	MFD_NPBSS_6_damper_open AT%I* : BOOL;
	MFD_NPBSS_6_damper_close AT%I* : BOOL;

	MFD_NPBSS_7_damper_open AT%I* : BOOL;
	MFD_NPBSS_7_damper_close AT%I* : BOOL;

	MFD_NPBSS_8_damper_open AT%I* : BOOL;
	MFD_NPBSS_8_damper_close AT%I* : BOOL;

	MFD_NPBSS_9_damper_open AT%I* : BOOL;
	MFD_NPBSS_9_damper_close AT%I* : BOOL;

	MFD_NPBSS_10_damper_open AT%I* : BOOL;
	MFD_NPBSS_10_damper_close AT%I* : BOOL;

(*************************************************************)
	common_alarm AT%Q* : BOOL;
	dcs_occupied AT%Q* : BOOL;

END_VAR
AHU_NPBSS_1_status_Filter(IN:=(NOT AHU_NPBSS_1_status AND AHU_NPBSS_1_latch),Q=>AHU_NPBSS_1_status_error);
AHU_NPBSS_1_trip_Filter(IN:=(AHU_NPBSS_1_trip AND AHU_NPBSS_1_latch),Q=>AHU_NPBSS_1_trip_error);
AHU_NPBSS_1_common_alarm := AHU_NPBSS_1_fire OR AHU_NPBSS_1_gas OR AHU_NPBSS_1_smoke OR AHU_NPBSS_1_status_error OR AHU_NPBSS_1_trip_error;


AHU_NPBSS_2_status_Filter(IN:=(NOT AHU_NPBSS_2_status AND AHU_NPBSS_2_latch),Q=>AHU_NPBSS_2_status_error);
AHU_NPBSS_2_trip_Filter(IN:=(AHU_NPBSS_2_trip AND AHU_NPBSS_2_latch),Q=>AHU_NPBSS_2_trip_error);
AHU_NPBSS_2_common_alarm := AHU_NPBSS_2_fire OR AHU_NPBSS_2_gas OR AHU_NPBSS_2_smoke OR AHU_NPBSS_2_status_error OR AHU_NPBSS_2_trip_error;


AHU_NPBSS_common_alarm := AHU_NPBSS_1_common_alarm OR AHU_NPBSS_2_common_alarm;
AHU_NPBSS_dcs_occupied := AHU_NPBSS_1_dcs_occupied OR AHU_NPBSS_2_dcs_occupied;

	FB_AHU_NPBSS(
	ON1:=AHU_NPBSS_1_trigger ,
	ON2:=AHU_NPBSS_2_trigger ,
	ON3:=FALSE ,
	status_error_1:= AHU_NPBSS_1_status_error,
	status_error_2:=AHU_NPBSS_2_status_error ,
	status_error_3:=FALSE ,
	trip_error_1:=AHU_NPBSS_1_trip_error ,
	trip_error_2:=AHU_NPBSS_2_trip_error ,
	trip_error_3:=FALSE ,
	Latch1:=AHU_NPBSS_1_latch ,
	Latch2:=AHU_NPBSS_2_latch ,
	Latch3:=AHU_NPBSS_dummy ,
	DcsOccupied_1=>AHU_NPBSS_1_dcs_occupied ,
	DcsOccupied_2=>AHU_NPBSS_2_dcs_occupied ,
	DcsOccupied_3=> );


(*********************************)

EF_NPBSS_1_status_Filter(IN:=(NOT EF_NPBSS_1_status AND EF_NPBSS_1_latch),Q=>EF_NPBSS_1_status_error);
EF_NPBSS_1_trip_Filter(IN:=(EF_NPBSS_1_trip AND EF_NPBSS_1_latch),Q=>EF_NPBSS_1_trip_error);
EF_NPBSS_1_common_alarm := EF_NPBSS_1_status_error OR EF_NPBSS_1_trip_error;

EF_NPBSS_2_status_Filter(IN:=(NOT EF_NPBSS_2_status AND EF_NPBSS_2_latch),Q=>EF_NPBSS_2_status_error);
EF_NPBSS_2_trip_Filter(IN:=(EF_NPBSS_2_trip AND EF_NPBSS_2_latch),Q=>EF_NPBSS_2_trip_error);
EF_NPBSS_2_common_alarm := EF_NPBSS_2_status_error OR EF_NPBSS_2_trip_error;


EF_NPBSS_common_alarm := EF_NPBSS_1_common_alarm OR EF_NPBSS_2_common_alarm;
EF_NPBSS_dcs_occupied := EF_NPBSS_1_dcs_occupied OR EF_NPBSS_2_dcs_occupied;

	FB_EF_NPBSS(
	ON1:=EF_NPBSS_1_trigger ,
	ON2:=EF_NPBSS_2_trigger ,
	ON3:=FALSE ,
	status_error_1:= EF_NPBSS_1_status_error,
	status_error_2:=EF_NPBSS_2_status_error ,
	status_error_3:=FALSE ,
	trip_error_1:=EF_NPBSS_1_trip_error ,
	trip_error_2:=EF_NPBSS_2_trip_error ,
	trip_error_3:=FALSE ,
	Latch1:=EF_NPBSS_1_latch ,
	Latch2:=EF_NPBSS_2_latch ,
	Latch3:=EF_NPBSS_dummy ,
	DcsOccupied_1=>EF_NPBSS_1_dcs_occupied ,
	DcsOccupied_2=>EF_NPBSS_2_dcs_occupied ,
	DcsOccupied_3=> );

(******************************************************)

EF_NPBSS_3_latch := TRUE;

EF_NPBSS_3_status_Filter(IN:=(NOT EF_NPBSS_3_status AND EF_NPBSS_3_latch),Q=>EF_NPBSS_3_status_error);
EF_NPBSS_3_trip_Filter(IN:=(EF_NPBSS_3_trip AND EF_NPBSS_3_latch),Q=>EF_NPBSS_3_trip_error);
EF_NPBSS_3_common_alarm := EF_NPBSS_3_status_error OR EF_NPBSS_3_trip_error;

(******************************************************)

EDH_NPBSS_3_on_status := AHU_NPBSS_dcs_occupied;

EDH_NPBSS_3_hightemp_error := EDH_NPBSS_3_high_temp;
EDH_NPBSS_3_common_alarm := EDH_NPBSS_3_hightemp_error;

FB_EDH_NPBSS_3(on_status:= EDH_NPBSS_3_on_status , flow_status:= EDH_NPBSS_3_flow_status , high_temp:= EDH_NPBSS_3_high_temp);

(****************************************************)

common_alarm := AHU_NPBSS_common_alarm OR EF_NPBSS_common_alarm OR EF_NPBSS_3_common_alarm OR EDH_NPBSS_3_common_alarm;
dcs_occupied := AHU_NPBSS_dcs_occupied OR EF_NPBSS_dcs_occupied;
END_PROGRAM

(* POU JettyOperation, ST *)
PROGRAM JettyOperation
VAR
	AHU_JOR_common_alarm : BOOL;
	AHU_JOR_dcs_occupied : BOOL;

	AHU_JOR_dummy : BOOL;
	FB_AHU_JOR: Flowchart_3_4_CTRL;

	AHU_JOR_1_status AT%I* : BOOL;
	AHU_JOR_1_trip AT%I* : BOOL;
	AHU_JOR_1_mode AT%I* : BOOL;
	AHU_JOR_1_belt AT%I* : BOOL;
	AHU_JOR_1_fire AT%I* : BOOL;
	AHU_JOR_1_gas AT%I* : BOOL;
	AHU_JOR_1_smoke AT%I* : BOOL;

	AHU_JOR_1_trigger : BOOL;
	AHU_JOR_1_latch : BOOL;
	AHU_JOR_1_common_alarm : BOOL;
	AHU_JOR_1_status_error : BOOL;
	AHU_JOR_1_trip_error : BOOL;
	AHU_JOR_1_dcs_occupied : BOOL;

	AHU_JOR_1_status_Filter : ErrorFilter;
	AHU_JOR_1_trip_Filter : ErrorFilter;


	AHU_JOR_2_status AT%I* : BOOL;
	AHU_JOR_2_trip AT%I* : BOOL;
	AHU_JOR_2_mode AT%I* : BOOL;
	AHU_JOR_2_belt AT%I* : BOOL;
	AHU_JOR_2_fire AT%I* : BOOL;
	AHU_JOR_2_gas AT%I* : BOOL;
	AHU_JOR_2_smoke AT%I* : BOOL;

	AHU_JOR_2_trigger : BOOL;
	AHU_JOR_2_latch : BOOL;
	AHU_JOR_2_common_alarm : BOOL;
	AHU_JOR_2_status_error : BOOL;
	AHU_JOR_2_trip_error : BOOL;
	AHU_JOR_2_dcs_occupied : BOOL;

	AHU_JOR_2_status_Filter : ErrorFilter;
	AHU_JOR_2_trip_Filter : ErrorFilter;

(**************************************************)

	EF_JOR_common_alarm : BOOL;
	EF_JOR_dcs_occupied : BOOL;

	EF_JOR_dummy : BOOL;
	FB_EF_JOR: Flowchart_3_4_CTRL;

	EF_JOR_1A_status AT%I* : BOOL;
	EF_JOR_1A_trip AT%I* : BOOL;
	EF_JOR_1A_mode AT%I* : BOOL;

	EF_JOR_1A_trigger : BOOL;
	EF_JOR_1A_latch : BOOL;
	EF_JOR_1A_common_alarm : BOOL;
	EF_JOR_1A_status_error : BOOL;
	EF_JOR_1A_trip_error : BOOL;
	EF_JOR_1A_dcs_occupied : BOOL;

	EF_JOR_1A_status_Filter : ErrorFilter;
	EF_JOR_1A_trip_Filter : ErrorFilter;


	EF_JOR_1B_status AT%I* : BOOL;
	EF_JOR_1B_trip AT%I* : BOOL;
	EF_JOR_1B_mode AT%I* : BOOL;

	EF_JOR_1B_trigger : BOOL;
	EF_JOR_1B_latch : BOOL;
	EF_JOR_1B_common_alarm : BOOL;
	EF_JOR_1B_status_error : BOOL;
	EF_JOR_1B_trip_error : BOOL;
	EF_JOR_1B_dcs_occupied : BOOL;

	EF_JOR_1B_status_Filter : ErrorFilter;
	EF_JOR_1B_trip_Filter : ErrorFilter;

(*************************************************************)

	EF_JOR_common_alarm_2 : BOOL;
	EF_JOR_dcs_occupied_2 : BOOL;


	FB_EF_JOR_2: Flowchart_7;

	EF_JOR_2_status AT%I* : BOOL;
	EF_JOR_2_trip AT%I* : BOOL;
	EF_JOR_2_mode AT%I* : BOOL;

	EF_JOR_2_trigger : BOOL;
	EF_JOR_2_latch : BOOL;
	EF_JOR_2_common_alarm : BOOL;
	EF_JOR_2_status_error : BOOL;
	EF_JOR_2_trip_error : BOOL;
	EF_JOR_2_dcs_occupied : BOOL;

	EF_JOR_2_status_Filter : ErrorFilter;
	EF_JOR_2_trip_Filter : ErrorFilter;


	FB_EF_JOR_3: Flowchart_7;

	EF_JOR_3_status AT%I* : BOOL;
	EF_JOR_3_trip AT%I* : BOOL;
	EF_JOR_3_mode AT%I* : BOOL;

	EF_JOR_3_trigger : BOOL;
	EF_JOR_3_latch : BOOL;
	EF_JOR_3_common_alarm : BOOL;
	EF_JOR_3_status_error : BOOL;
	EF_JOR_3_trip_error : BOOL;
	EF_JOR_3_dcs_occupied : BOOL;

	EF_JOR_3_status_Filter : ErrorFilter;
	EF_JOR_3_trip_Filter : ErrorFilter;

(************************************************************)

	EF_JOR_common_alarm_3 : BOOL;


	EF_JOR_4A_status AT%I* : BOOL;
	EF_JOR_4A_trip AT%I* : BOOL;
	EF_JOR_4A_mode AT%I* : BOOL;

	EF_JOR_4A_trigger : BOOL;
	EF_JOR_4A_latch : BOOL;
	EF_JOR_4A_common_alarm : BOOL;
	EF_JOR_4A_status_error : BOOL;
	EF_JOR_4A_trip_error : BOOL;
	EF_JOR_4A_dcs_occupied : BOOL;

	EF_JOR_4A_status_Filter : ErrorFilter;
	EF_JOR_4A_trip_Filter : ErrorFilter;



	EF_JOR_4B_status AT%I* : BOOL;
	EF_JOR_4B_trip AT%I* : BOOL;
	EF_JOR_4B_mode AT%I* : BOOL;

	EF_JOR_4B_trigger : BOOL;
	EF_JOR_4B_latch : BOOL;
	EF_JOR_4B_common_alarm : BOOL;
	EF_JOR_4B_status_error : BOOL;
	EF_JOR_4B_trip_error : BOOL;
	EF_JOR_4B_dcs_occupied : BOOL;

	EF_JOR_4B_status_Filter : ErrorFilter;
	EF_JOR_4B_trip_Filter : ErrorFilter;


	EF_JOR_5_status AT%I* : BOOL;
	EF_JOR_5_trip AT%I* : BOOL;
	EF_JOR_5_mode AT%I* : BOOL;

	EF_JOR_5_trigger : BOOL;
	EF_JOR_5_latch : BOOL;
	EF_JOR_5_common_alarm : BOOL;
	EF_JOR_5_status_error : BOOL;
	EF_JOR_5_trip_error : BOOL;
	EF_JOR_5_dcs_occupied : BOOL;

	EF_JOR_5_status_Filter : ErrorFilter;
	EF_JOR_5_trip_Filter : ErrorFilter;

(********************************************************************)


	FB_EDH_JOR_1: Flowchart_5_6;
	EDH_JOR_1_on_status : BOOL;
	EDH_JOR_1_flow_status AT%I* : BOOL;
	EDH_JOR_1_high_temp AT%I* : BOOL;

	EDH_JOR_1_common_alarm : BOOL;
	EDH_JOR_1_hightemp_error : BOOL;

(*********************************************************)

	MD_JOR_1A_damper_open AT%I* : BOOL;
	MD_JOR_1A_damper_close AT%I* : BOOL;

	MD_JOR_1B_damper_open AT%I* : BOOL;
	MD_JOR_1B_damper_close AT%I* : BOOL;

	MD_JOR_1C_damper_open AT%I* : BOOL;
	MD_JOR_1C_damper_close AT%I* : BOOL;

	MD_JOR_2A_damper_open AT%I* : BOOL;
	MD_JOR_2A_damper_close AT%I* : BOOL;

	MD_JOR_2B_damper_open AT%I* : BOOL;
	MD_JOR_2B_damper_close AT%I* : BOOL;

	MD_JOR_3A_damper_open AT%I* : BOOL;
	MD_JOR_3A_damper_close AT%I* : BOOL;

(***********************************************************)


	MFD_JOR_1_damper_open AT%I* : BOOL;
	MFD_JOR_1_damper_close AT%I* : BOOL;

	MFD_JOR_2_damper_open AT%I* : BOOL;
	MFD_JOR_2_damper_close AT%I* : BOOL;

	MFD_JOR_3_damper_open AT%I* : BOOL;
	MFD_JOR_3_damper_close AT%I* : BOOL;

	MFD_JOR_4_damper_open AT%I* : BOOL;
	MFD_JOR_4_damper_close AT%I* : BOOL;

	MFD_JOR_5_damper_open AT%I* : BOOL;
	MFD_JOR_5_damper_close AT%I* : BOOL;

	MFD_JOR_6_damper_open AT%I* : BOOL;
	MFD_JOR_6_damper_close AT%I* : BOOL;

	MFD_JOR_7_damper_open AT%I* : BOOL;
	MFD_JOR_7_damper_close AT%I* : BOOL;

(**********************************************************)

	common_alarm AT%Q* : BOOL;
	dcs_occupied AT%Q* : BOOL;

END_VAR
AHU_JOR_1_status_Filter(IN:=(NOT AHU_JOR_1_status AND AHU_JOR_1_latch),Q=>AHU_JOR_1_status_error);
AHU_JOR_1_trip_Filter(IN:=(AHU_JOR_1_trip AND AHU_JOR_1_latch),Q=>AHU_JOR_1_trip_error);
AHU_JOR_1_common_alarm := AHU_JOR_1_fire OR AHU_JOR_1_gas OR AHU_JOR_1_smoke OR AHU_JOR_1_status_error OR AHU_JOR_1_trip_error;



AHU_JOR_2_status_Filter(IN:=(NOT AHU_JOR_2_status AND AHU_JOR_2_latch),Q=>AHU_JOR_2_status_error);
AHU_JOR_2_trip_Filter(IN:=(AHU_JOR_2_trip AND AHU_JOR_2_latch),Q=>AHU_JOR_2_trip_error);
AHU_JOR_2_common_alarm := AHU_JOR_2_fire OR AHU_JOR_2_gas OR AHU_JOR_2_smoke OR AHU_JOR_2_status_error OR AHU_JOR_2_trip_error;


AHU_JOR_common_alarm := AHU_JOR_1_common_alarm OR AHU_JOR_2_common_alarm;
AHU_JOR_dcs_occupied := AHU_JOR_1_dcs_occupied OR AHU_JOR_2_dcs_occupied;

	FB_AHU_JOR(
	ON1:=AHU_JOR_1_trigger ,
	ON2:=AHU_JOR_2_trigger ,
	ON3:=FALSE ,
	status_error_1:= AHU_JOR_1_status_error,
	status_error_2:=AHU_JOR_2_status_error ,
	status_error_3:=FALSE ,
	trip_error_1:=AHU_JOR_1_trip_error ,
	trip_error_2:=AHU_JOR_2_trip_error ,
	trip_error_3:=FALSE ,
	Latch1:=AHU_JOR_1_latch ,
	Latch2:=AHU_JOR_2_latch ,
	Latch3:=AHU_JOR_dummy ,
	DcsOccupied_1=>AHU_JOR_1_dcs_occupied ,
	DcsOccupied_2=>AHU_JOR_2_dcs_occupied ,
	DcsOccupied_3=> );

(*************************************************************)


EF_JOR_1A_status_Filter(IN:=(NOT EF_JOR_1A_status AND EF_JOR_1A_latch),Q=>EF_JOR_1A_status_error);
EF_JOR_1A_trip_Filter(IN:=(EF_JOR_1A_trip AND EF_JOR_1A_latch),Q=>EF_JOR_1A_trip_error);
EF_JOR_1A_common_alarm := EF_JOR_1A_status_error OR EF_JOR_1A_trip_error;

EF_JOR_1B_status_Filter(IN:=(NOT EF_JOR_1B_status AND EF_JOR_1B_latch),Q=>EF_JOR_1B_status_error);
EF_JOR_1B_trip_Filter(IN:=(EF_JOR_1B_trip AND EF_JOR_1B_latch),Q=>EF_JOR_1B_trip_error);
EF_JOR_1B_common_alarm := EF_JOR_1B_status_error OR EF_JOR_1B_trip_error;


EF_JOR_common_alarm := EF_JOR_1A_common_alarm OR EF_JOR_1B_common_alarm;
EF_JOR_dcs_occupied := EF_JOR_1A_dcs_occupied OR EF_JOR_1B_dcs_occupied;

	FB_EF_JOR(
	ON1:=EF_JOR_1A_trigger ,
	ON2:=EF_JOR_1B_trigger ,
	ON3:=FALSE ,
	status_error_1:= EF_JOR_1A_status_error,
	status_error_2:=EF_JOR_1B_status_error ,
	status_error_3:=FALSE ,
	trip_error_1:=EF_JOR_1A_trip_error ,
	trip_error_2:=EF_JOR_1B_trip_error ,
	trip_error_3:=FALSE ,
	Latch1:=EF_JOR_1A_latch ,
	Latch2:=EF_JOR_1B_latch ,
	Latch3:=EF_JOR_dummy ,
	DcsOccupied_1=>EF_JOR_1A_dcs_occupied ,
	DcsOccupied_2=>EF_JOR_1B_dcs_occupied ,
	DcsOccupied_3=> );

(***********************************************************)



EF_JOR_2_status_Filter(IN:=(NOT EF_JOR_2_status AND EF_JOR_2_latch),Q=>EF_JOR_2_status_error);
EF_JOR_2_trip_Filter(IN:=(EF_JOR_2_trip AND EF_JOR_2_latch),Q=>EF_JOR_2_trip_error);
EF_JOR_2_common_alarm := EF_JOR_2_status_error OR EF_JOR_2_trip_error;


FB_EF_JOR_2(
Trigger:=EF_JOR_2_trigger ,
Latch:=EF_JOR_2_latch ,
DCS_Occupied=>EF_JOR_2_dcs_occupied );




EF_JOR_3_status_Filter(IN:=(NOT EF_JOR_3_status AND EF_JOR_3_latch),Q=>EF_JOR_3_status_error);
EF_JOR_3_trip_Filter(IN:=(EF_JOR_3_trip AND EF_JOR_3_latch),Q=>EF_JOR_3_trip_error);
EF_JOR_3_common_alarm := EF_JOR_3_status_error OR EF_JOR_3_trip_error;


FB_EF_JOR_3(
Trigger:=EF_JOR_3_trigger ,
Latch:=EF_JOR_3_latch ,
DCS_Occupied=>EF_JOR_3_dcs_occupied );


EF_JOR_common_alarm_2:=EF_JOR_2_common_alarm OR EF_JOR_3_common_alarm;
EF_JOR_dcs_occupied_2:=EF_JOR_2_dcs_occupied OR EF_JOR_3_dcs_occupied;

(************************************************************)

EF_JOR_4A_status_Filter(IN:=(NOT EF_JOR_4A_status AND EF_JOR_4A_latch),Q=>EF_JOR_4A_status_error);
EF_JOR_4A_trip_Filter(IN:=(EF_JOR_4A_trip AND EF_JOR_4A_latch),Q=>EF_JOR_4A_trip_error);
EF_JOR_4A_common_alarm := EF_JOR_4A_status_error OR EF_JOR_4A_trip_error;

EF_JOR_4B_status_Filter(IN:=(NOT EF_JOR_4B_status AND EF_JOR_4B_latch),Q=>EF_JOR_4B_status_error);
EF_JOR_4B_trip_Filter(IN:=(EF_JOR_4B_trip AND EF_JOR_4B_latch),Q=>EF_JOR_4B_trip_error);
EF_JOR_4B_common_alarm := EF_JOR_4B_status_error OR EF_JOR_4B_trip_error;


EF_JOR_5_status_Filter(IN:=(NOT EF_JOR_5_status AND EF_JOR_5_latch),Q=>EF_JOR_5_status_error);
EF_JOR_5_trip_Filter(IN:=(EF_JOR_5_trip AND EF_JOR_5_latch),Q=>EF_JOR_5_trip_error);
EF_JOR_5_common_alarm := EF_JOR_5_status_error OR EF_JOR_5_trip_error;


EF_JOR_common_alarm_3:=EF_JOR_4A_common_alarm OR EF_JOR_4B_common_alarm OR EF_JOR_5_common_alarm;

(****************************************************************************************)

EDH_JOR_1_on_status := AHU_JOR_common_alarm;
EDH_JOR_1_hightemp_error := EDH_JOR_1_high_temp;
EDH_JOR_1_common_alarm := EDH_JOR_1_hightemp_error;

FB_EDH_JOR_1(on_status:= EDH_JOR_1_on_status , flow_status:= EDH_JOR_1_flow_status , high_temp:= EDH_JOR_1_high_temp);

(****************************************************************************************)

common_alarm := EF_JOR_common_alarm OR AHU_JOR_common_alarm OR EF_JOR_common_alarm_2;
dcs_occupied := EF_JOR_dcs_occupied OR AHU_JOR_dcs_occupied OR EF_JOR_dcs_occupied_2 OR EF_JOR_common_alarm_3;
END_PROGRAM

(* POU JettySubStation, ST *)
PROGRAM JettySubStation
VAR
	AHU_JSS_common_alarm : BOOL;
	AHU_JSS_dcs_occupied : BOOL;

	AHU_JSS_dummy : BOOL;
	FB_AHU_JSS: Flowchart_3_4_CTRL;

	AHU_JSS_1_status AT%I* : BOOL;
	AHU_JSS_1_trip AT%I* : BOOL;
	AHU_JSS_1_mode AT%I* : BOOL;
	AHU_JSS_1_belt AT%I* : BOOL;
	AHU_JSS_1_fire AT%I* : BOOL;
	AHU_JSS_1_gas AT%I* : BOOL;
	AHU_JSS_1_smoke AT%I* : BOOL;

	AHU_JSS_1_trigger : BOOL;
	AHU_JSS_1_latch : BOOL;
	AHU_JSS_1_common_alarm : BOOL;
	AHU_JSS_1_status_error : BOOL;
	AHU_JSS_1_trip_error : BOOL;
	AHU_JSS_1_dcs_occupied : BOOL;

	AHU_JSS_1_status_Filter : ErrorFilter;
	AHU_JSS_1_trip_Filter : ErrorFilter;


	AHU_JSS_2_status AT%I* : BOOL;
	AHU_JSS_2_trip AT%I* : BOOL;
	AHU_JSS_2_mode AT%I* : BOOL;
	AHU_JSS_2_belt AT%I* : BOOL;
	AHU_JSS_2_fire AT%I* : BOOL;
	AHU_JSS_2_gas AT%I* : BOOL;
	AHU_JSS_2_smoke AT%I* : BOOL;

	AHU_JSS_2_trigger : BOOL;
	AHU_JSS_2_latch : BOOL;
	AHU_JSS_2_common_alarm : BOOL;
	AHU_JSS_2_status_error : BOOL;
	AHU_JSS_2_trip_error : BOOL;
	AHU_JSS_2_dcs_occupied : BOOL;

	AHU_JSS_2_status_Filter : ErrorFilter;
	AHU_JSS_2_trip_Filter : ErrorFilter;

(**************************************************)

	EF_JSS_common_alarm : BOOL;
	EF_JSS_dcs_occupied : BOOL;

	EF_JSS_dummy : BOOL;
	FB_EF_JSS: Flowchart_3_4_CTRL;

	EF_JSS_1A_status AT%I* : BOOL;
	EF_JSS_1A_trip AT%I* : BOOL;
	EF_JSS_1A_mode AT%I* : BOOL;

	EF_JSS_1A_trigger : BOOL;
	EF_JSS_1A_latch : BOOL;
	EF_JSS_1A_common_alarm : BOOL;
	EF_JSS_1A_status_error : BOOL;
	EF_JSS_1A_trip_error : BOOL;
	EF_JSS_1A_dcs_occupied : BOOL;

	EF_JSS_1A_status_Filter : ErrorFilter;
	EF_JSS_1A_trip_Filter : ErrorFilter;


	EF_JSS_1B_status AT%I* : BOOL;
	EF_JSS_1B_trip AT%I* : BOOL;
	EF_JSS_1B_mode AT%I* : BOOL;

	EF_JSS_1B_trigger : BOOL;
	EF_JSS_1B_latch : BOOL;
	EF_JSS_1B_common_alarm : BOOL;
	EF_JSS_1B_status_error : BOOL;
	EF_JSS_1B_trip_error : BOOL;
	EF_JSS_1B_dcs_occupied : BOOL;

	EF_JSS_1B_status_Filter : ErrorFilter;
	EF_JSS_1B_trip_Filter : ErrorFilter;

(*************************************************************)

	EF_JSS_common_alarm_2 : BOOL;

	EF_JSS_2_status AT%I* : BOOL;
	EF_JSS_2_trip AT%I* : BOOL;
	EF_JSS_2_mode AT%I* : BOOL;

	EF_JSS_2_trigger : BOOL;
	EF_JSS_2_latch : BOOL;
	EF_JSS_2_common_alarm : BOOL;
	EF_JSS_2_status_error : BOOL;
	EF_JSS_2_trip_error : BOOL;
	EF_JSS_2_dcs_occupied : BOOL;

	EF_JSS_2_status_Filter : ErrorFilter;
	EF_JSS_2_trip_Filter : ErrorFilter;


(********************************************************************)


	FB_EDH_JSS_1: Flowchart_5_6;
	EDH_JSS_1_on_status : BOOL;
	EDH_JSS_1_flow_status AT%I* : BOOL;
	EDH_JSS_1_high_temp AT%I* : BOOL;

	EDH_JSS_1_common_alarm : BOOL;
	EDH_JSS_1_hightemp_error : BOOL;

(*********************************************************)

	MD_JSS_1A_damper_open AT%I* : BOOL;
	MD_JSS_1A_damper_close AT%I* : BOOL;

	MD_JSS_1B_damper_open AT%I* : BOOL;
	MD_JSS_1B_damper_close AT%I* : BOOL;

	MD_JSS_1C_damper_open AT%I* : BOOL;
	MD_JSS_1C_damper_close AT%I* : BOOL;

	MD_JSS_1D_damper_open AT%I* : BOOL;
	MD_JSS_1D_damper_close AT%I* : BOOL;


(***********************************************************)


	MFD_JSS_1_damper_open AT%I* : BOOL;
	MFD_JSS_1_damper_close AT%I* : BOOL;

	MFD_JSS_2_damper_open AT%I* : BOOL;
	MFD_JSS_2_damper_close AT%I* : BOOL;

	MFD_JSS_3_damper_open AT%I* : BOOL;
	MFD_JSS_3_damper_close AT%I* : BOOL;

	MFD_JSS_4_damper_open AT%I* : BOOL;
	MFD_JSS_4_damper_close AT%I* : BOOL;

	MFD_JSS_5_damper_open AT%I* : BOOL;
	MFD_JSS_5_damper_close AT%I* : BOOL;

	MFD_JSS_6_damper_open AT%I* : BOOL;
	MFD_JSS_6_damper_close AT%I* : BOOL;

	MFD_JSS_7_damper_open AT%I* : BOOL;
	MFD_JSS_7_damper_close AT%I* : BOOL;

	MFD_JSS_8_damper_open AT%I* : BOOL;
	MFD_JSS_8_damper_close AT%I* : BOOL;

	MFD_JSS_9_damper_open AT%I* : BOOL;
	MFD_JSS_9_damper_close AT%I* : BOOL;

(****************************************************************)
	common_alarm AT%Q* : BOOL;
	dcs_occupied AT%Q* : BOOL;



END_VAR
AHU_JSS_1_status_Filter(IN:=(NOT AHU_JSS_1_status AND AHU_JSS_1_latch),Q=>AHU_JSS_1_status_error);
AHU_JSS_1_trip_Filter(IN:=(AHU_JSS_1_trip AND AHU_JSS_1_latch),Q=>AHU_JSS_1_trip_error);
AHU_JSS_1_common_alarm := AHU_JSS_1_fire OR AHU_JSS_1_gas OR AHU_JSS_1_smoke OR AHU_JSS_1_status_error OR AHU_JSS_1_trip_error;



AHU_JSS_2_status_Filter(IN:=(NOT AHU_JSS_2_status AND AHU_JSS_2_latch),Q=>AHU_JSS_2_status_error);
AHU_JSS_2_trip_Filter(IN:=(AHU_JSS_2_trip AND AHU_JSS_2_latch),Q=>AHU_JSS_2_trip_error);
AHU_JSS_2_common_alarm := AHU_JSS_2_fire OR AHU_JSS_2_gas OR AHU_JSS_2_smoke OR AHU_JSS_2_status_error OR AHU_JSS_2_trip_error;


AHU_JSS_common_alarm := AHU_JSS_1_common_alarm OR AHU_JSS_2_common_alarm;
AHU_JSS_dcs_occupied := AHU_JSS_1_dcs_occupied OR AHU_JSS_2_dcs_occupied;

	FB_AHU_JSS(
	ON1:=AHU_JSS_1_trigger ,
	ON2:=AHU_JSS_2_trigger ,
	ON3:=FALSE ,
	status_error_1:= AHU_JSS_1_status_error,
	status_error_2:=AHU_JSS_2_status_error ,
	status_error_3:=FALSE ,
	trip_error_1:=AHU_JSS_1_trip_error ,
	trip_error_2:=AHU_JSS_2_trip_error ,
	trip_error_3:=FALSE ,
	Latch1:=AHU_JSS_1_latch ,
	Latch2:=AHU_JSS_2_latch ,
	Latch3:=AHU_JSS_dummy ,
	DcsOccupied_1=>AHU_JSS_1_dcs_occupied ,
	DcsOccupied_2=>AHU_JSS_2_dcs_occupied ,
	DcsOccupied_3=> );

(*************************************************************)


EF_JSS_1A_status_Filter(IN:=(NOT EF_JSS_1A_status AND EF_JSS_1A_latch),Q=>EF_JSS_1A_status_error);
EF_JSS_1A_trip_Filter(IN:=(EF_JSS_1A_trip AND EF_JSS_1A_latch),Q=>EF_JSS_1A_trip_error);
EF_JSS_1A_common_alarm := EF_JSS_1A_status_error OR EF_JSS_1A_trip_error;

EF_JSS_1B_status_Filter(IN:=(NOT EF_JSS_1B_status AND EF_JSS_1B_latch),Q=>EF_JSS_1B_status_error);
EF_JSS_1B_trip_Filter(IN:=(EF_JSS_1B_trip AND EF_JSS_1B_latch),Q=>EF_JSS_1B_trip_error);
EF_JSS_1B_common_alarm := EF_JSS_1B_status_error OR EF_JSS_1B_trip_error;


EF_JSS_common_alarm := EF_JSS_1A_common_alarm OR EF_JSS_1B_common_alarm;
EF_JSS_dcs_occupied := EF_JSS_1A_dcs_occupied OR EF_JSS_1B_dcs_occupied;

	FB_EF_JSS(
	ON1:=EF_JSS_1A_trigger ,
	ON2:=EF_JSS_1B_trigger ,
	ON3:=FALSE ,
	status_error_1:= EF_JSS_1A_status_error,
	status_error_2:=EF_JSS_1B_status_error ,
	status_error_3:=FALSE ,
	trip_error_1:=EF_JSS_1A_trip_error ,
	trip_error_2:=EF_JSS_1B_trip_error ,
	trip_error_3:=FALSE ,
	Latch1:=EF_JSS_1A_latch ,
	Latch2:=EF_JSS_1B_latch ,
	Latch3:=EF_JSS_dummy ,
	DcsOccupied_1=>EF_JSS_1A_dcs_occupied ,
	DcsOccupied_2=>EF_JSS_1B_dcs_occupied ,
	DcsOccupied_3=> );

(***********************************************************)

EF_JSS_2_latch :=TRUE;

EF_JSS_2_status_Filter(IN:=(NOT EF_JSS_2_status AND EF_JSS_2_latch),Q=>EF_JSS_2_status_error);
EF_JSS_2_trip_Filter(IN:=(EF_JSS_2_trip AND EF_JSS_2_latch),Q=>EF_JSS_2_trip_error);
EF_JSS_2_common_alarm := EF_JSS_2_status_error OR EF_JSS_2_trip_error;

EF_JSS_common_alarm_2 := EF_JSS_2_common_alarm;


(****************************************************************************************)
EDH_JSS_1_on_status := AHU_JSS_dcs_occupied;

EDH_JSS_1_hightemp_error := EDH_JSS_1_high_temp;
EDH_JSS_1_common_alarm := EDH_JSS_1_hightemp_error;

FB_EDH_JSS_1(on_status:= EDH_JSS_1_on_status , flow_status:= EDH_JSS_1_flow_status , high_temp:= EDH_JSS_1_high_temp);

(**************************************************************************************)

common_alarm := AHU_JSS_common_alarm OR EF_JSS_common_alarm OR EF_JSS_common_alarm_2 OR EDH_JSS_1_common_alarm;
dcs_occupied := AHU_JSS_dcs_occupied OR EF_JSS_dcs_occupied;
END_PROGRAM

(* POU OfficeSubStation, ST *)
PROGRAM OfficeSubStation
VAR
	AHU_OFFSS_common_alarm : BOOL;
	AHU_OFFSS_dcs_occupied : BOOL;

	AHU_OFFSS_dummy : BOOL;
	FB_AHU_OFFSS: Flowchart_3_4_CTRL;

	AHU_OFFSS_1_status AT%I* : BOOL;
	AHU_OFFSS_1_trip AT%I* : BOOL;
	AHU_OFFSS_1_mode AT%I* : BOOL;
	AHU_OFFSS_1_belt AT%I* : BOOL;
	AHU_OFFSS_1_fire AT%I* : BOOL;
	AHU_OFFSS_1_gas AT%I* : BOOL;
	AHU_OFFSS_1_smoke AT%I* : BOOL;

	AHU_OFFSS_1_trigger : BOOL;
	AHU_OFFSS_1_latch : BOOL;
	AHU_OFFSS_1_common_alarm : BOOL;
	AHU_OFFSS_1_status_error : BOOL;
	AHU_OFFSS_1_trip_error : BOOL;
	AHU_OFFSS_1_dcs_occupied : BOOL;

	AHU_OFFSS_1_status_Filter : ErrorFilter;
	AHU_OFFSS_1_trip_Filter : ErrorFilter;


	AHU_OFFSS_2_status AT%I* : BOOL;
	AHU_OFFSS_2_trip AT%I* : BOOL;
	AHU_OFFSS_2_mode AT%I* : BOOL;
	AHU_OFFSS_2_belt AT%I* : BOOL;
	AHU_OFFSS_2_fire AT%I* : BOOL;
	AHU_OFFSS_2_gas AT%I* : BOOL;
	AHU_OFFSS_2_smoke AT%I* : BOOL;

	AHU_OFFSS_2_trigger : BOOL;
	AHU_OFFSS_2_latch : BOOL;
	AHU_OFFSS_2_common_alarm : BOOL;
	AHU_OFFSS_2_status_error : BOOL;
	AHU_OFFSS_2_trip_error : BOOL;
	AHU_OFFSS_2_dcs_occupied : BOOL;

	AHU_OFFSS_2_status_Filter : ErrorFilter;
	AHU_OFFSS_2_trip_Filter : ErrorFilter;

(**************************************************)

	EF_OFFSS_common_alarm : BOOL;
	EF_OFFSS_dcs_occupied : BOOL;

	EF_OFFSS_dummy : BOOL;
	FB_EF_OFFSS: Flowchart_3_4_CTRL;

	EF_OFFSS_1A_status AT%I* : BOOL;
	EF_OFFSS_1A_trip AT%I* : BOOL;
	EF_OFFSS_1A_mode AT%I* : BOOL;

	EF_OFFSS_1A_trigger : BOOL;
	EF_OFFSS_1A_latch : BOOL;
	EF_OFFSS_1A_common_alarm : BOOL;
	EF_OFFSS_1A_status_error : BOOL;
	EF_OFFSS_1A_trip_error : BOOL;
	EF_OFFSS_1A_dcs_occupied : BOOL;

	EF_OFFSS_1A_status_Filter : ErrorFilter;
	EF_OFFSS_1A_trip_Filter : ErrorFilter;


	EF_OFFSS_1B_status AT%I* : BOOL;
	EF_OFFSS_1B_trip AT%I* : BOOL;
	EF_OFFSS_1B_mode AT%I* : BOOL;

	EF_OFFSS_1B_trigger : BOOL;
	EF_OFFSS_1B_latch : BOOL;
	EF_OFFSS_1B_common_alarm : BOOL;
	EF_OFFSS_1B_status_error : BOOL;
	EF_OFFSS_1B_trip_error : BOOL;
	EF_OFFSS_1B_dcs_occupied : BOOL;

	EF_OFFSS_1B_status_Filter : ErrorFilter;
	EF_OFFSS_1B_trip_Filter : ErrorFilter;

(*************************************************************)

	EF_OFFSS_common_alarm_2 : BOOL;

	EF_OFFSS_2A_status AT%I* : BOOL;
	EF_OFFSS_2A_trip AT%I* : BOOL;
	EF_OFFSS_2A_mode AT%I* : BOOL;

	EF_OFFSS_2A_trigger : BOOL;
	EF_OFFSS_2A_latch : BOOL;
	EF_OFFSS_2A_common_alarm : BOOL;
	EF_OFFSS_2A_status_error : BOOL;
	EF_OFFSS_2A_trip_error : BOOL;
	EF_OFFSS_2A_dcs_occupied : BOOL;

	EF_OFFSS_2A_status_Filter : ErrorFilter;
	EF_OFFSS_2A_trip_Filter : ErrorFilter;


	EF_OFFSS_2B_status AT%I* : BOOL;
	EF_OFFSS_2B_trip AT%I* : BOOL;
	EF_OFFSS_2B_mode AT%I* : BOOL;

	EF_OFFSS_2B_trigger : BOOL;
	EF_OFFSS_2B_latch : BOOL;
	EF_OFFSS_2B_common_alarm : BOOL;
	EF_OFFSS_2B_status_error : BOOL;
	EF_OFFSS_2B_trip_error : BOOL;
	EF_OFFSS_2B_dcs_occupied : BOOL;

	EF_OFFSS_2B_status_Filter : ErrorFilter;
	EF_OFFSS_2B_trip_Filter : ErrorFilter;

(********************************************************************)


	FB_EDH_OFFSS_1: Flowchart_5_6;
	EDH_OFFSS_1_on_status : BOOL;
	EDH_OFFSS_1_flow_status AT%I* : BOOL;
	EDH_OFFSS_1_high_temp AT%I* : BOOL;

	EDH_OFFSS_1_common_alarm : BOOL;
	EDH_OFFSS_1_hightemp_error : BOOL;

(*********************************************************)

	MD_OFFSS_1A_damper_open AT%I* : BOOL;
	MD_OFFSS_1A_damper_close AT%I* : BOOL;

	MD_OFFSS_1B_damper_open AT%I* : BOOL;
	MD_OFFSS_1B_damper_close AT%I* : BOOL;

	MD_OFFSS_1C_damper_open AT%I* : BOOL;
	MD_OFFSS_1C_damper_close AT%I* : BOOL;

	MD_OFFSS_1D_damper_open AT%I* : BOOL;
	MD_OFFSS_1D_damper_close AT%I* : BOOL;

	MD_OFFSS_1E_damper_open AT%I* : BOOL;
	MD_OFFSS_1E_damper_close AT%I* : BOOL;


(***********************************************************)


	MFD_OFFSS_1_damper_open AT%I* : BOOL;
	MFD_OFFSS_1_damper_close AT%I* : BOOL;

	MFD_OFFSS_2_damper_open AT%I* : BOOL;
	MFD_OFFSS_2_damper_close AT%I* : BOOL;

	MFD_OFFSS_3_damper_open AT%I* : BOOL;
	MFD_OFFSS_3_damper_close AT%I* : BOOL;

	MFD_OFFSS_4_damper_open AT%I* : BOOL;
	MFD_OFFSS_4_damper_close AT%I* : BOOL;

	MFD_OFFSS_5_damper_open AT%I* : BOOL;
	MFD_OFFSS_5_damper_close AT%I* : BOOL;

	MFD_OFFSS_6_damper_open AT%I* : BOOL;
	MFD_OFFSS_6_damper_close AT%I* : BOOL;

	MFD_OFFSS_7_damper_open AT%I* : BOOL;
	MFD_OFFSS_7_damper_close AT%I* : BOOL;

	MFD_OFFSS_8_damper_open AT%I* : BOOL;
	MFD_OFFSS_8_damper_close AT%I* : BOOL;

	MFD_OFFSS_9_damper_open AT%I* : BOOL;
	MFD_OFFSS_9_damper_close AT%I* : BOOL;

(************************************************************************)

	common_alarm AT%Q* : BOOL;
	dcs_occupied AT%Q* : BOOL;

END_VAR
AHU_OFFSS_1_status_Filter(IN:=(NOT AHU_OFFSS_1_status AND AHU_OFFSS_1_latch),Q=>AHU_OFFSS_1_status_error);
AHU_OFFSS_1_trip_Filter(IN:=(AHU_OFFSS_1_trip AND AHU_OFFSS_1_latch),Q=>AHU_OFFSS_1_trip_error);
AHU_OFFSS_1_common_alarm := AHU_OFFSS_1_fire OR AHU_OFFSS_1_gas OR AHU_OFFSS_1_smoke OR AHU_OFFSS_1_status_error OR AHU_OFFSS_1_trip_error;



AHU_OFFSS_2_status_Filter(IN:=(NOT AHU_OFFSS_2_status AND AHU_OFFSS_2_latch),Q=>AHU_OFFSS_2_status_error);
AHU_OFFSS_2_trip_Filter(IN:=(AHU_OFFSS_2_trip AND AHU_OFFSS_2_latch),Q=>AHU_OFFSS_2_trip_error);
AHU_OFFSS_2_common_alarm := AHU_OFFSS_2_fire OR AHU_OFFSS_2_gas OR AHU_OFFSS_2_smoke OR AHU_OFFSS_2_status_error OR AHU_OFFSS_2_trip_error;


AHU_OFFSS_common_alarm := AHU_OFFSS_1_common_alarm OR AHU_OFFSS_2_common_alarm;
AHU_OFFSS_dcs_occupied := AHU_OFFSS_1_dcs_occupied OR AHU_OFFSS_2_dcs_occupied;

	FB_AHU_OFFSS(
	ON1:=AHU_OFFSS_1_trigger ,
	ON2:=AHU_OFFSS_2_trigger ,
	ON3:=FALSE ,
	status_error_1:= AHU_OFFSS_1_status_error,
	status_error_2:=AHU_OFFSS_2_status_error ,
	status_error_3:=FALSE ,
	trip_error_1:=AHU_OFFSS_1_trip_error ,
	trip_error_2:=AHU_OFFSS_2_trip_error ,
	trip_error_3:=FALSE ,
	Latch1:=AHU_OFFSS_1_latch ,
	Latch2:=AHU_OFFSS_2_latch ,
	Latch3:=AHU_OFFSS_dummy ,
	DcsOccupied_1=>AHU_OFFSS_1_dcs_occupied ,
	DcsOccupied_2=>AHU_OFFSS_2_dcs_occupied ,
	DcsOccupied_3=> );

(*************************************************************)


EF_OFFSS_1A_status_Filter(IN:=(NOT EF_OFFSS_1A_status AND EF_OFFSS_1A_latch),Q=>EF_OFFSS_1A_status_error);
EF_OFFSS_1A_trip_Filter(IN:=(EF_OFFSS_1A_trip AND EF_OFFSS_1A_latch),Q=>EF_OFFSS_1A_trip_error);
EF_OFFSS_1A_common_alarm := EF_OFFSS_1A_status_error OR EF_OFFSS_1A_trip_error;

EF_OFFSS_1B_status_Filter(IN:=(NOT EF_OFFSS_1B_status AND EF_OFFSS_1B_latch),Q=>EF_OFFSS_1B_status_error);
EF_OFFSS_1B_trip_Filter(IN:=(EF_OFFSS_1B_trip AND EF_OFFSS_1B_latch),Q=>EF_OFFSS_1B_trip_error);
EF_OFFSS_1B_common_alarm := EF_OFFSS_1B_status_error OR EF_OFFSS_1B_trip_error;


EF_OFFSS_common_alarm := EF_OFFSS_1A_common_alarm OR EF_OFFSS_1B_common_alarm;
EF_OFFSS_dcs_occupied := EF_OFFSS_1A_dcs_occupied OR EF_OFFSS_1B_dcs_occupied;

	FB_EF_OFFSS(
	ON1:=EF_OFFSS_1A_trigger ,
	ON2:=EF_OFFSS_1B_trigger ,
	ON3:=FALSE ,
	status_error_1:= EF_OFFSS_1A_status_error,
	status_error_2:=EF_OFFSS_1B_status_error ,
	status_error_3:=FALSE ,
	trip_error_1:=EF_OFFSS_1A_trip_error ,
	trip_error_2:=EF_OFFSS_1B_trip_error ,
	trip_error_3:=FALSE ,
	Latch1:=EF_OFFSS_1A_latch ,
	Latch2:=EF_OFFSS_1B_latch ,
	Latch3:=EF_OFFSS_dummy ,
	DcsOccupied_1=>EF_OFFSS_1A_dcs_occupied ,
	DcsOccupied_2=>EF_OFFSS_1B_dcs_occupied ,
	DcsOccupied_3=> );

(***********************************************************)

EF_OFFSS_2A_latch :=TRUE;

EF_OFFSS_2A_status_Filter(IN:=(NOT EF_OFFSS_2A_status AND EF_OFFSS_2A_latch),Q=>EF_OFFSS_2A_status_error);
EF_OFFSS_2A_trip_Filter(IN:=(EF_OFFSS_2A_trip AND EF_OFFSS_2A_latch),Q=>EF_OFFSS_2A_trip_error);
EF_OFFSS_2A_common_alarm := EF_OFFSS_2A_status_error OR EF_OFFSS_2A_trip_error;


EF_OFFSS_2B_latch :=TRUE;

EF_OFFSS_2B_status_Filter(IN:=(NOT EF_OFFSS_2B_status AND EF_OFFSS_2B_latch),Q=>EF_OFFSS_2B_status_error);
EF_OFFSS_2B_trip_Filter(IN:=(EF_OFFSS_2B_trip AND EF_OFFSS_2B_latch),Q=>EF_OFFSS_2B_trip_error);
EF_OFFSS_2B_common_alarm := EF_OFFSS_2B_status_error OR EF_OFFSS_2B_trip_error;

EF_OFFSS_common_alarm_2 := EF_OFFSS_2A_common_alarm OR EF_OFFSS_2B_common_alarm;


(****************************************************************************************)
EDH_OFFSS_1_on_status :=AHU_OFFSS_dcs_occupied;

EDH_OFFSS_1_hightemp_error := EDH_OFFSS_1_high_temp;
EDH_OFFSS_1_common_alarm := EDH_OFFSS_1_hightemp_error;

FB_EDH_OFFSS_1(on_status:= EDH_OFFSS_1_on_status , flow_status:= EDH_OFFSS_1_flow_status , high_temp:= EDH_OFFSS_1_high_temp);

(***************************************************************************************)

common_alarm := AHU_OFFSS_common_alarm OR EF_OFFSS_common_alarm OR EF_OFFSS_common_alarm_2 OR EDH_OFFSS_1_common_alarm;
dcs_occupied := AHU_OFFSS_dcs_occupied OR EF_OFFSS_dcs_occupied;
END_PROGRAM

(* POU GarbageCan/CCB_GroundFloor_CFC, CFC *)
PROGRAM CCB_GroundFloor_CFC
VAR
	AHU_CCBG_01_02_03: Flowchart_1_2_SingleButton;

	bAHUCCBG1_On: BOOL;
	bAHUCCBG2_On: BOOL;
	bAHUCCBG3_On: BOOL;

	AHUCCBG1_DcsOccupied: BOOL;
	AHUCCBG1_StatusError: BOOL;
	AHUCCBG1_TripError: BOOL;
	AHUCCBG2_DcsOccupied: BOOL;
	AHUCCBG2_StatusError: BOOL;
	AHUCCBG2_TripError: BOOL;
	AHUCCBG3_DcsOccupied: BOOL;
	AHUCCBG3_StatusError: BOOL;
	AHUCCBG3_TripError: BOOL;

	AHUCCBG_CommonAlarm AT %Q*: BOOL;
	AHUCCBG_DcsOccupied AT %Q*: BOOL;

	AHUCCBG1_Smoke AT%I* : BOOL;
	AHUCCBG1_Fire AT%I*:BOOL;
	AHUCCBG1_Gas AT%I*:BOOL;

	AHUCCBG2_Smoke AT%I* : BOOL;
	AHUCCBG2_Fire AT%I*:BOOL;
	AHUCCBG2_Gas AT%I*:BOOL;

	AHUCCBG3_Smoke AT%I* : BOOL;
	AHUCCBG3_Fire AT%I*:BOOL;
	AHUCCBG3_Gas AT%I*:BOOL;

	EEF_CCB_1_2: Flowchart_3_4_SingleButton;

	bAHU1_Battery: BOOL;
	bAHU2_Battery: BOOL;
	AHU1Battery_DcsOccupied: BOOL;
	AHU1Battery_StatusError: BOOL;
	AHU1Battery_TripError: BOOL;
	AHU2Battery_DcsOccupied: BOOL;
	AHU2Battery_StatusError: BOOL;
	AHU2Battery_TripError: BOOL;
	AHUBattery_CommonAlarm AT%Q*: BOOL;
	AHUBattery_DcsOccupied AT%Q*: BOOL;

	TEF_CCB_01: Flowchart_7;
	bFanOn: BOOL;
	FAN_DcsOccupied AT%Q*: BOOL;
	FAN_Battery_StatusError: BOOL;
	FAN_Battery_TripError: BOOL;
	FAN_CommonAlarm AT%Q*: BOOL;


	EH_CCB_01: Flowchart_5_6;
	HEATERCCB1_CommonAlarm AT %Q*: BOOL;
	HEATERCCB1_FlowStatus: BOOL;
	HEATERCCB1_TEMP: INT;
	HEATERCCB1_STAGE1 AT %Q*: BOOL;
	HEATERCCB1_STAGE2 AT %Q*: BOOL;
	HEATERCCB1_STAGE3 AT %Q*: BOOL;

	EH_CCB_02: Flowchart_5_6;
	HEATERCCB2_CommonAlarm AT %Q*: BOOL;
	HEATERCCB2_FlowStatus: BOOL;
	HEATERCCB2_TEMP: INT;
	HEATERCCB2_STAGE1 AT %Q*: BOOL;
	HEATERCCB2_STAGE2 AT %Q*: BOOL;
	HEATERCCB2_STAGE3 AT %Q*: BOOL;

	Damper_MD_CCBG_1 AT%I* : BOOL;
	Damper_MD_CCBG_2 AT%I* : BOOL;
	Damper_MD_CCBG_3 AT%I* : BOOL;
	Damper_MD_CCBG_4 AT%I* : BOOL;

	Damper_MD_EF_07A  AT%I* : BOOL;
	Damper_MD_EF_07B  AT%I* : BOOL;
	Damper_MD_EF_08  AT%I* : BOOL;

	FireDAmper_MD_CCB_01 AT%I* : BOOL;
	FireDAmper_MD_CCB_02 AT%I* : BOOL;
	FireDAmper_MD_CCB_03 AT%I* : BOOL;
	FireDAmper_MD_CCB_04 AT%I* : BOOL;
	FireDAmper_MD_CCB_05 AT%I* : BOOL;
	FireDAmper_MD_CCB_06 AT%I* : BOOL;
	FireDAmper_MD_CCB_07 AT%I* : BOOL;
	FireDAmper_MD_CCB_08 AT%I* : BOOL;
	FireDAmper_MD_CCB_09 AT%I* : BOOL;
	FireDAmper_MD_CCB_10 AT%I* : BOOL;

END_VAR
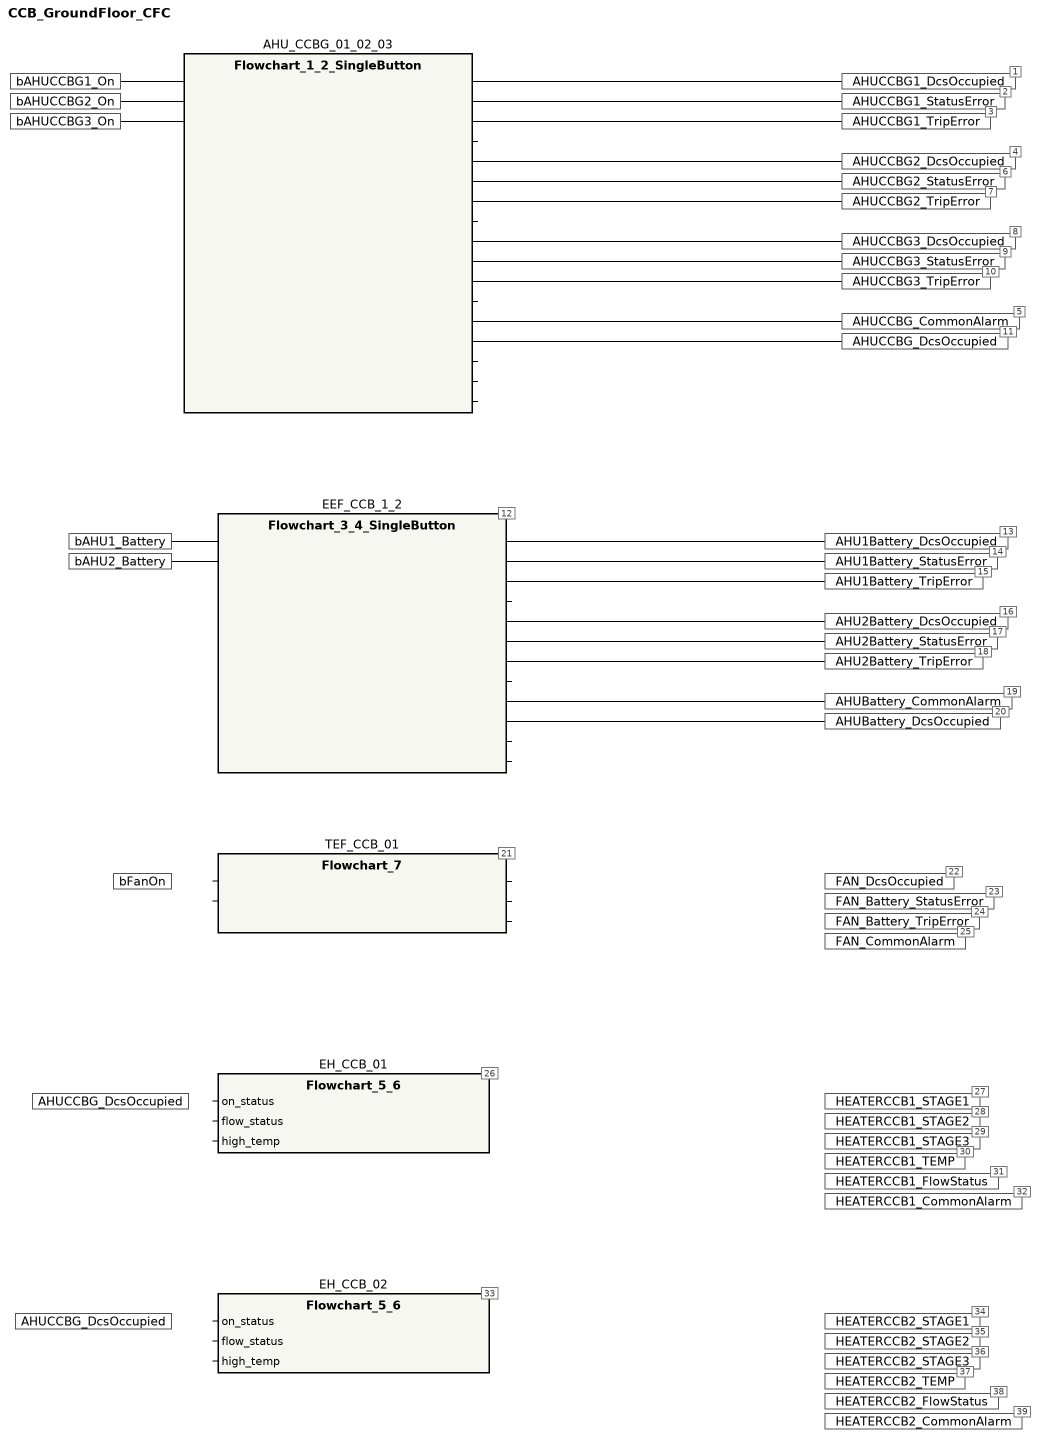
_CFC_ (* Continuous Function Chart, elements in execution order *)
#0 AHU_CCBG_01_02_03:Flowchart_1_2_SingleButton(bAHUCCBG1_On, bAHUCCBG2_On, bAHUCCBG3_On)
#1 AHUCCBG1_DcsOccupied <= #0.out 1
#2 AHUCCBG1_StatusError <= #0.out 2
#3 AHUCCBG1_TripError <= #0.out 3
#4 AHUCCBG2_DcsOccupied <= #0.out 5
#5 AHUCCBG_CommonAlarm <= #0.out 13
#6 AHUCCBG2_StatusError <= #0.out 6
#7 AHUCCBG2_TripError <= #0.out 7
#8 AHUCCBG3_DcsOccupied <= #0.out 9
#9 AHUCCBG3_StatusError <= #0.out 10
#10 AHUCCBG3_TripError <= #0.out 11
#11 AHUCCBG_DcsOccupied <= #0.out 14
#12 EEF_CCB_1_2:Flowchart_3_4_SingleButton(bAHU1_Battery, bAHU2_Battery)
#13 AHU1Battery_DcsOccupied <= #12.out 1
#14 AHU1Battery_StatusError <= #12.out 2
#15 AHU1Battery_TripError <= #12.out 3
#16 AHU2Battery_DcsOccupied <= #12.out 5
#17 AHU2Battery_StatusError <= #12.out 6
#18 AHU2Battery_TripError <= #12.out 7
#19 AHUBattery_CommonAlarm <= #12.out 9
#20 AHUBattery_DcsOccupied <= #12.out 10
unconnected input bFanOn
#21 TEF_CCB_01:Flowchart_7(-, -)
#22 FAN_DcsOccupied <= -
#23 FAN_Battery_StatusError <= -
#24 FAN_Battery_TripError <= -
#25 FAN_CommonAlarm <= -
unconnected input AHUCCBG_DcsOccupied
#26 EH_CCB_01:Flowchart_5_6(on_status: -, flow_status: -, high_temp: -)
#27 HEATERCCB1_STAGE1 <= -
#28 HEATERCCB1_STAGE2 <= -
#29 HEATERCCB1_STAGE3 <= -
#30 HEATERCCB1_TEMP <= -
#31 HEATERCCB1_FlowStatus <= -
#32 HEATERCCB1_CommonAlarm <= -
unconnected input AHUCCBG_DcsOccupied
#33 EH_CCB_02:Flowchart_5_6(on_status: -, flow_status: -, high_temp: -)
#34 HEATERCCB2_STAGE1 <= -
#35 HEATERCCB2_STAGE2 <= -
#36 HEATERCCB2_STAGE3 <= -
#37 HEATERCCB2_TEMP <= -
#38 HEATERCCB2_FlowStatus <= -
#39 HEATERCCB2_CommonAlarm <= -
_END_CFC_
END_PROGRAM

(* POU GarbageCan/Flowchart_1_2_SingleButton, CFC *)
FUNCTION_BLOCK Flowchart_1_2_SingleButton
VAR_INPUT
END_VAR
VAR_OUTPUT
	AHU1_DcsOccupied : BOOL;
	AHU1_StatusError  : BOOL;
	AHU1_TripError : BOOL;
	bAHU1_Error: BOOL;

	AHU2_DcsOccupied : BOOL;
	AHU2_StatusError  : BOOL;
	AHU2_TripError : BOOL;
	bAHU2_Error: BOOL;

	AHU3_DcsOccupied : BOOL;
	AHU3_StatusError : BOOL;
	AHU3_TripError : BOOL;
	bAHU3_Error: BOOL;

	AHU_CommonAlarm:BOOL;
	AHU_DCSOccupied:BOOL;
END_VAR
VAR

	bAHU1_Status AT %I*: BOOL;
	bAHU1_Trip AT %I*: BOOL;
	bAHU1_Relay AT %Q*: BOOL;
	Status_timer_1: TON;
	Error_timer_1: TOF;
	OnRtrigAHU1: R_TRIG;
	OffRtrigAHU1: R_TRIG;


	bAHU2_Status AT %I*: BOOL;
	bAHU2_Trip AT %I*: BOOL;
	bAHU2_Relay AT %Q*: BOOL;
	Status_timer_2: TON;
	Error_timer_2: TOF;
	OnRtrigAHU2: R_TRIG;
	OffRtrigAHU2: R_TRIG;


	bAHU3_Status AT %I*: BOOL;
	bAHU3_Trip AT %I*: BOOL;
	bAHU3_Relay AT %Q*: BOOL;
	Status_timer_3: TON;
	Error_timer_3: TOF;
	OnRtrigAHU3: R_TRIG;
	OffRtrigAHU3: R_TRIG;


	AHU1_Reset: TON;
	AHU2_Reset: TON;
	AHU3_Reset: TON;
END_VAR
VAR_IN_OUT
	bAHU1_On: BOOL;
	bAHU2_On: BOOL;
	bAHU3_On: BOOL;
END_VAR
VAR (* helpers for the ST form of the networks *)
	_t14 : BOOL;
	_t31 : BOOL;
	_t34 : BOOL;
	_t65 : BOOL;
	_t137 : BOOL;
	_t150 : BOOL;
	_t147 : BOOL;
	_t152 : BOOL;
	_t208 : BOOL;
	_t176 : BOOL;
	_t189 : BOOL;
	_t186 : BOOL;
	_t191 : BOOL;
END_VAR
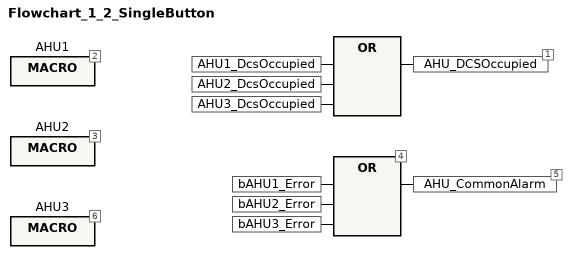
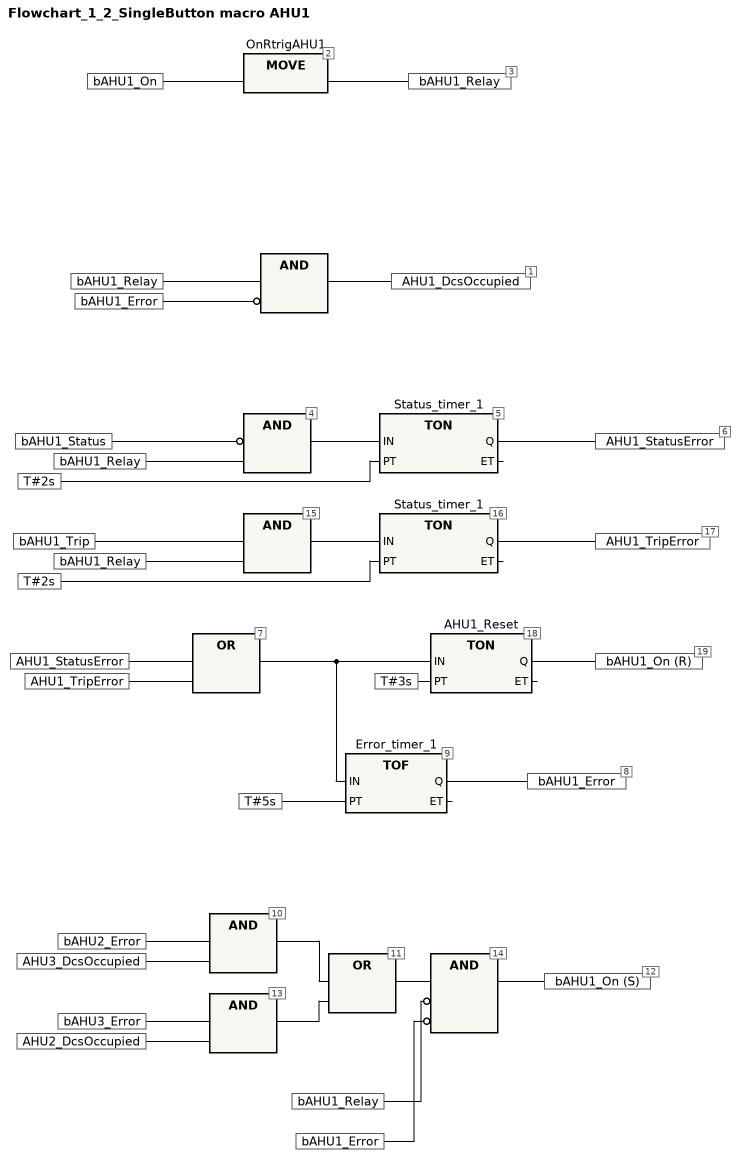
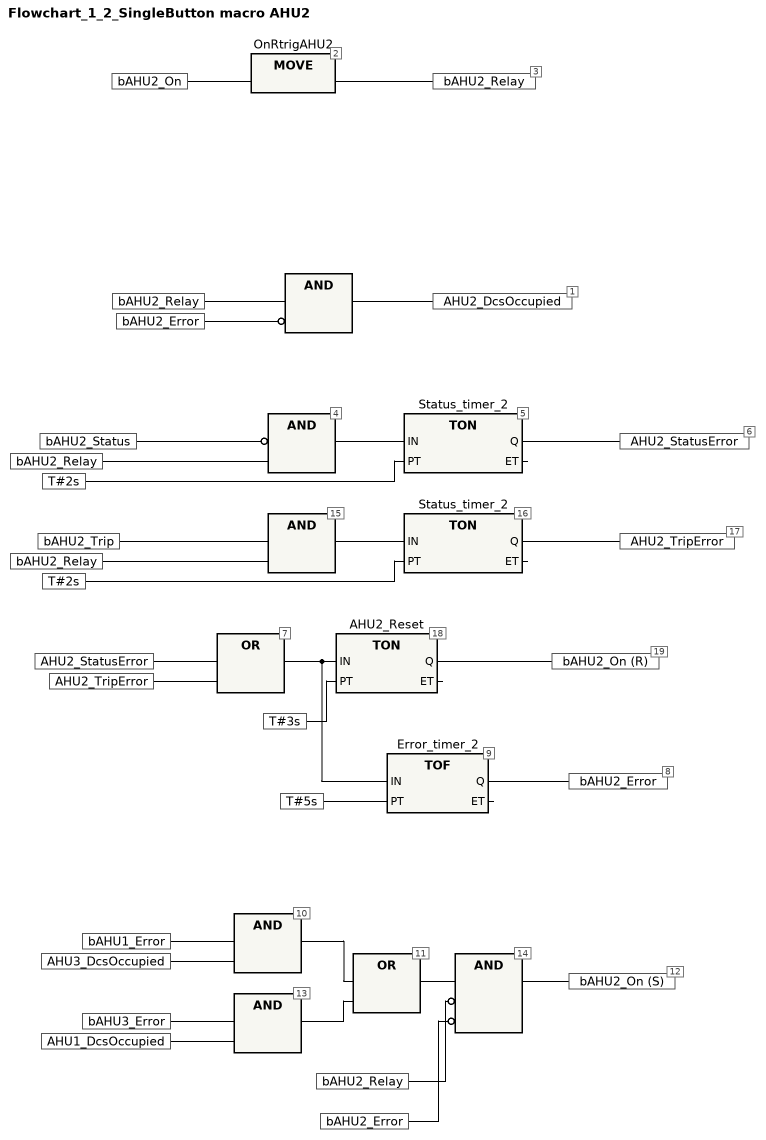
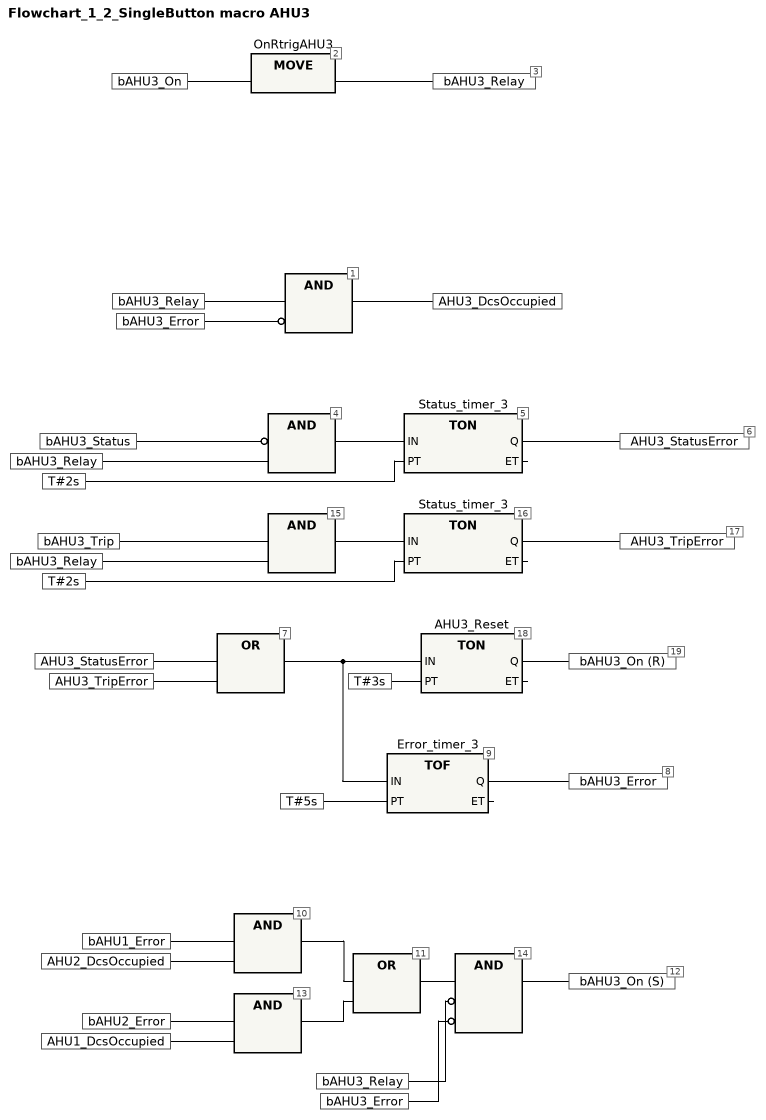
_CFC_ (* Continuous Function Chart, elements in execution order *)
#0 OR(AHU1_DcsOccupied, AHU2_DcsOccupied, AHU3_DcsOccupied)
#1 AHU_DCSOccupied <= #0
#2 MACRO AHU1()
	#3 AND(bAHU1_Relay, NOT bAHU1_Error)
	#4 AHU1_DcsOccupied <= #3
	#5 OnRtrigAHU1:MOVE(bAHU1_On)
	#6 bAHU1_Relay <= #5
	#7 AND(NOT bAHU1_Status, bAHU1_Relay)
	#8 Status_timer_1:TON(IN: #7, PT: T#2s)
	#9 AHU1_StatusError <= #8.Q
	#10 OR(AHU1_StatusError, AHU1_TripError)
	#11 bAHU1_Error <= #12.Q
	#12 Error_timer_1:TOF(IN: #10, PT: T#5s)
	#13 AND(bAHU2_Error, AHU3_DcsOccupied)
	#14 OR(#13, #16)
	#15 S bAHU1_On <= #17
	#16 AND(bAHU3_Error, AHU2_DcsOccupied)
	#17 AND(#14, NOT bAHU1_Relay, NOT bAHU1_Error)
	#18 AND(bAHU1_Trip, bAHU1_Relay)
	#19 Status_timer_1:TON(IN: #18, PT: T#2s)
	#20 AHU1_TripError <= #19.Q
	#21 AHU1_Reset:TON(IN: #10, PT: T#3s)
	#22 R bAHU1_On <= #21.Q
END_MACRO
#23 MACRO AHU2()
	#24 AND(bAHU2_Relay, NOT bAHU2_Error)
	#25 AHU2_DcsOccupied <= #24
	#26 OnRtrigAHU2:MOVE(bAHU2_On)
	#27 bAHU2_Relay <= #26
	#28 AND(NOT bAHU2_Status, bAHU2_Relay)
	#29 Status_timer_2:TON(IN: #28, PT: T#2s)
	#30 AHU2_StatusError <= #29.Q
	#31 OR(AHU2_StatusError, AHU2_TripError)
	#32 bAHU2_Error <= #33.Q
	#33 Error_timer_2:TOF(IN: #31, PT: T#5s)
	#34 AND(bAHU1_Error, AHU3_DcsOccupied)
	#35 OR(#34, #37)
	#36 S bAHU2_On <= #38
	#37 AND(bAHU3_Error, AHU1_DcsOccupied)
	#38 AND(#35, NOT bAHU2_Relay, NOT bAHU2_Error)
	#39 AND(bAHU2_Trip, bAHU2_Relay)
	#40 Status_timer_2:TON(IN: #39, PT: T#2s)
	#41 AHU2_TripError <= #40.Q
	#42 AHU2_Reset:TON(IN: #31, PT: T#3s)
	#43 R bAHU2_On <= #42.Q
END_MACRO
#44 OR(bAHU1_Error, bAHU2_Error, bAHU3_Error)
#45 AHU_CommonAlarm <= #44
#46 MACRO AHU3()
	#47 AHU3_DcsOccupied <= #48
	#48 AND(bAHU3_Relay, NOT bAHU3_Error)
	#49 OnRtrigAHU3:MOVE(bAHU3_On)
	#50 bAHU3_Relay <= #49
	#51 AND(NOT bAHU3_Status, bAHU3_Relay)
	#52 Status_timer_3:TON(IN: #51, PT: T#2s)
	#53 AHU3_StatusError <= #52.Q
	#54 OR(AHU3_StatusError, AHU3_TripError)
	#55 bAHU3_Error <= #56.Q
	#56 Error_timer_3:TOF(IN: #54, PT: T#5s)
	#57 AND(bAHU1_Error, AHU2_DcsOccupied)
	#58 OR(#57, #60)
	#59 S bAHU3_On <= #61
	#60 AND(bAHU2_Error, AHU1_DcsOccupied)
	#61 AND(#58, NOT bAHU3_Relay, NOT bAHU3_Error)
	#62 AND(bAHU3_Trip, bAHU3_Relay)
	#63 Status_timer_3:TON(IN: #62, PT: T#2s)
	#64 AHU3_TripError <= #63.Q
	#65 AHU3_Reset:TON(IN: #54, PT: T#3s)
	#66 R bAHU3_On <= #65.Q
END_MACRO
_END_CFC_
(* the same logic as Structured Text *)
AHU_DCSOccupied := AHU1_DcsOccupied OR AHU2_DcsOccupied OR AHU3_DcsOccupied;
(* macro AHU1 *)
AHU1_DcsOccupied := bAHU1_Relay AND NOT bAHU1_Error;
bAHU1_Relay := bAHU1_On;
Status_timer_1(IN := NOT bAHU1_Status AND bAHU1_Relay, PT := T#2s);
AHU1_StatusError := Status_timer_1.Q;
_t14 := AHU1_StatusError OR AHU1_TripError;
bAHU1_Error := Error_timer_1.Q;
Error_timer_1(IN := _t14, PT := T#5s);
_t34 := (bAHU2_Error AND AHU3_DcsOccupied) OR _t31;
IF _t65 THEN bAHU1_On := TRUE; END_IF;
_t31 := bAHU3_Error AND AHU2_DcsOccupied;
_t65 := _t34 AND NOT bAHU1_Relay AND NOT bAHU1_Error;
Status_timer_1(IN := bAHU1_Trip AND bAHU1_Relay, PT := T#2s);
AHU1_TripError := Status_timer_1.Q;
AHU1_Reset(IN := _t14, PT := T#3s);
IF AHU1_Reset.Q THEN bAHU1_On := FALSE; END_IF;
(* macro AHU2 *)
AHU2_DcsOccupied := bAHU2_Relay AND NOT bAHU2_Error;
bAHU2_Relay := bAHU2_On;
Status_timer_2(IN := NOT bAHU2_Status AND bAHU2_Relay, PT := T#2s);
AHU2_StatusError := Status_timer_2.Q;
_t137 := AHU2_StatusError OR AHU2_TripError;
bAHU2_Error := Error_timer_2.Q;
Error_timer_2(IN := _t137, PT := T#5s);
_t147 := (bAHU1_Error AND AHU3_DcsOccupied) OR _t150;
IF _t152 THEN bAHU2_On := TRUE; END_IF;
_t150 := bAHU3_Error AND AHU1_DcsOccupied;
_t152 := _t147 AND NOT bAHU2_Relay AND NOT bAHU2_Error;
Status_timer_2(IN := bAHU2_Trip AND bAHU2_Relay, PT := T#2s);
AHU2_TripError := Status_timer_2.Q;
AHU2_Reset(IN := _t137, PT := T#3s);
IF AHU2_Reset.Q THEN bAHU2_On := FALSE; END_IF;
AHU_CommonAlarm := bAHU1_Error OR bAHU2_Error OR bAHU3_Error;
(* macro AHU3 *)
AHU3_DcsOccupied := _t208;
_t208 := bAHU3_Relay AND NOT bAHU3_Error;
bAHU3_Relay := bAHU3_On;
Status_timer_3(IN := NOT bAHU3_Status AND bAHU3_Relay, PT := T#2s);
AHU3_StatusError := Status_timer_3.Q;
_t176 := AHU3_StatusError OR AHU3_TripError;
bAHU3_Error := Error_timer_3.Q;
Error_timer_3(IN := _t176, PT := T#5s);
_t186 := (bAHU1_Error AND AHU2_DcsOccupied) OR _t189;
IF _t191 THEN bAHU3_On := TRUE; END_IF;
_t189 := bAHU2_Error AND AHU1_DcsOccupied;
_t191 := _t186 AND NOT bAHU3_Relay AND NOT bAHU3_Error;
Status_timer_3(IN := bAHU3_Trip AND bAHU3_Relay, PT := T#2s);
AHU3_TripError := Status_timer_3.Q;
AHU3_Reset(IN := _t176, PT := T#3s);
IF AHU3_Reset.Q THEN bAHU3_On := FALSE; END_IF;
END_FUNCTION_BLOCK

(* POU GarbageCan/Flowchart_1_2, CFC *)
FUNCTION_BLOCK Flowchart_1_2
VAR_INPUT
	bAHU1_On: BOOL;
	bAHU1_Off: BOOL;


	bAHU2_On: BOOL;
	bAHU2_Off: BOOL;

	bAHU3_On: BOOL;
	bAHU3_Off: BOOL;
END_VAR
VAR_OUTPUT
	AHU1_DcsOccupied : BOOL;
	AHU1_StatusError  : BOOL;
	AHU1_TripError : BOOL;
	bAHU1_Error: BOOL;

	AHU2_DcsOccupied : BOOL;
	AHU2_StatusError  : BOOL;
	AHU2_TripError : BOOL;
	bAHU2_Error: BOOL;

	AHU3_DcsOccupied : BOOL;
	AHU3_StatusError : BOOL;
	AHU3_TripError : BOOL;
	bAHU3_Error: BOOL;

	AHU_CommonAlarm:BOOL;
	AHU_DCSOccupied:BOOL;
END_VAR
VAR


	bAHU1_Status AT %I*: BOOL;
	bAHU1_Trip AT %I*: BOOL;
	bAHU1_Relay AT %Q*: BOOL;
	Status_timer_1: TON;
	Error_timer_1: TOF;
	OnRtrigAHU1: R_TRIG;
	OffRtrigAHU1: R_TRIG;


	bAHU2_Status AT %I*: BOOL;
	bAHU2_Trip AT %I*: BOOL;
	bAHU2_Relay AT %Q*: BOOL;
	Status_timer_2: TON;
	Error_timer_2: TOF;
	OnRtrigAHU2: R_TRIG;
	OffRtrigAHU2: R_TRIG;


	bAHU3_Status AT %I*: BOOL;
	bAHU3_Trip AT %I*: BOOL;
	bAHU3_Relay AT %Q*: BOOL;
	Status_timer_3: TON;
	Error_timer_3: TOF;
	OnRtrigAHU3: R_TRIG;
	OffRtrigAHU3: R_TRIG;


	AHU1_Reset: TON;
	AHU2_Reset: TON;
	AHU3_Reset: TON;

END_VAR
VAR (* helpers for the ST form of the networks *)
	_t14 : BOOL;
	_t31 : BOOL;
	_t34 : BOOL;
	_t65 : BOOL;
	_t137 : BOOL;
	_t150 : BOOL;
	_t147 : BOOL;
	_t152 : BOOL;
	_t208 : BOOL;
	_t176 : BOOL;
	_t189 : BOOL;
	_t186 : BOOL;
	_t191 : BOOL;
END_VAR
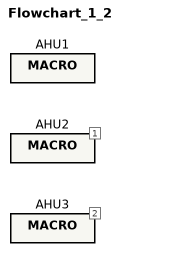
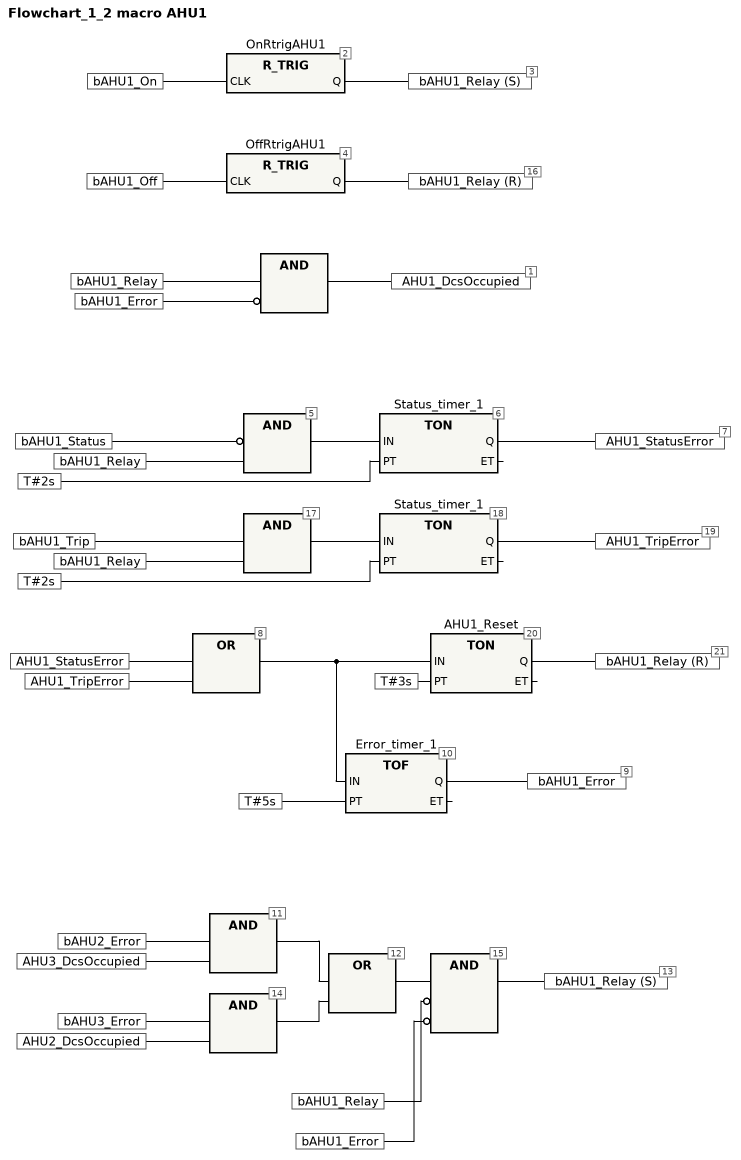
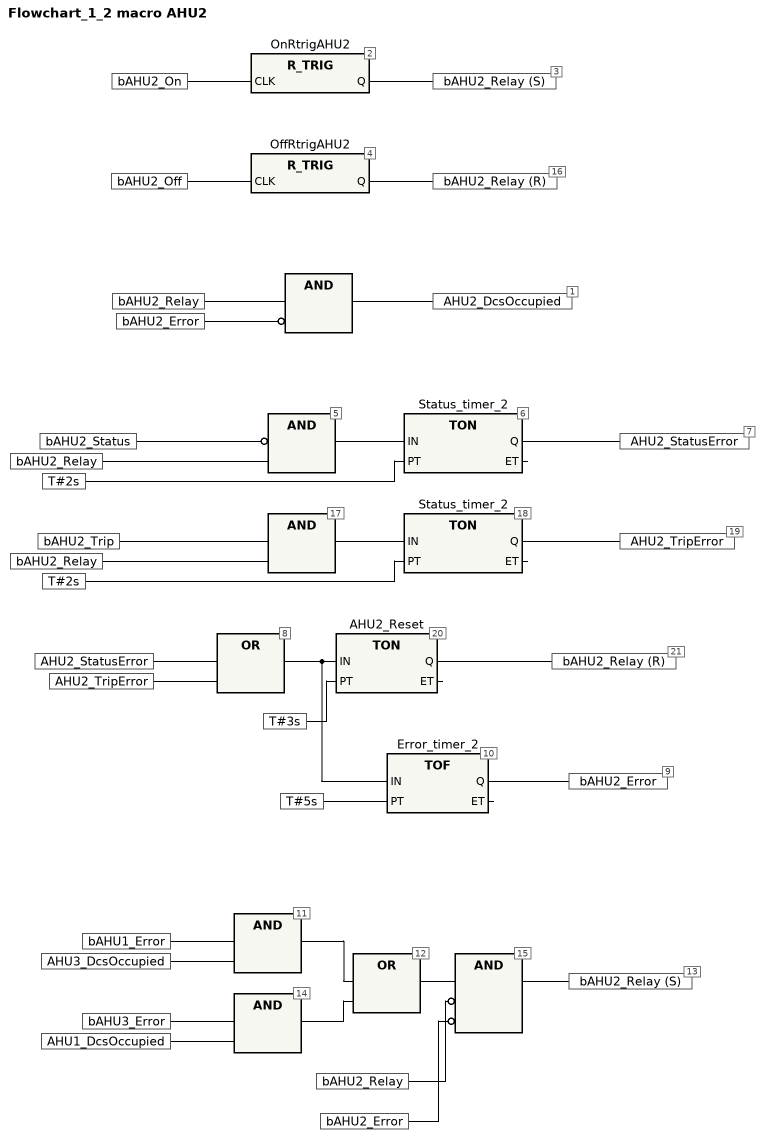
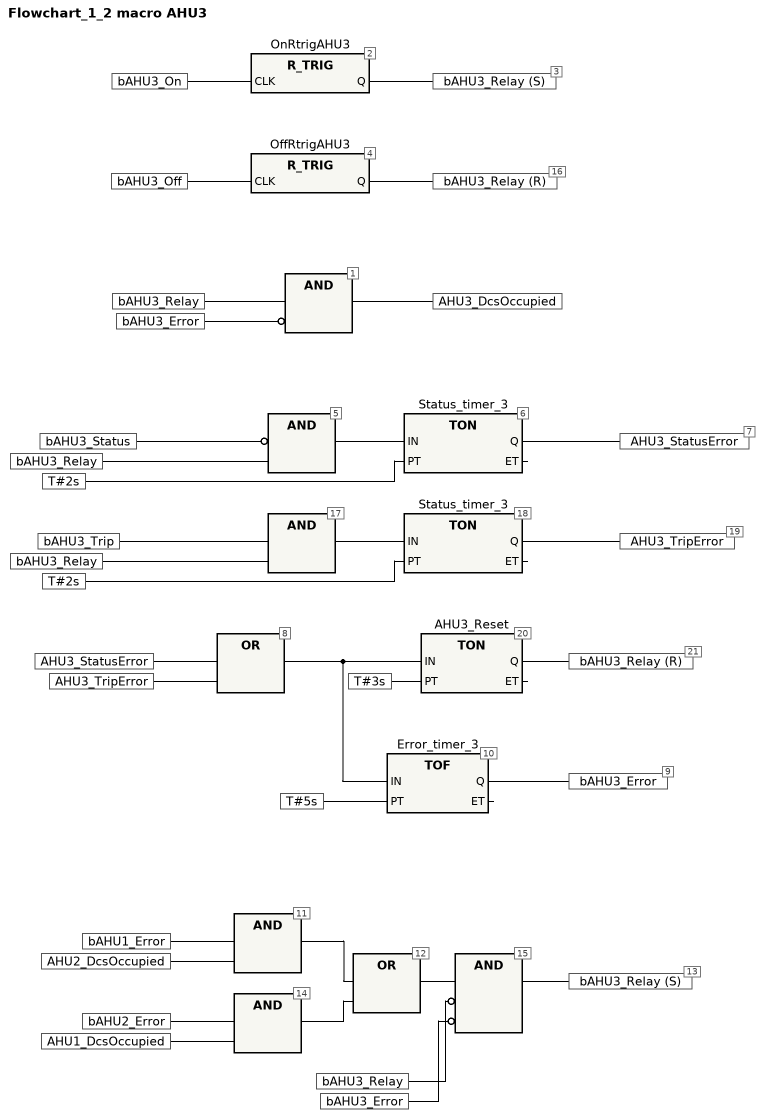
_CFC_ (* Continuous Function Chart, elements in execution order *)
#0 MACRO AHU1()
	#1 AND(bAHU1_Relay, NOT bAHU1_Error)
	#2 AHU1_DcsOccupied <= #1
	#3 OnRtrigAHU1:R_TRIG(CLK: bAHU1_On)
	#4 S bAHU1_Relay <= #3.Q
	#5 OffRtrigAHU1:R_TRIG(CLK: bAHU1_Off)
	#6 AND(NOT bAHU1_Status, bAHU1_Relay)
	#7 Status_timer_1:TON(IN: #6, PT: T#2s)
	#8 AHU1_StatusError <= #7.Q
	#9 OR(AHU1_StatusError, AHU1_TripError)
	#10 bAHU1_Error <= #11.Q
	#11 Error_timer_1:TOF(IN: #9, PT: T#5s)
	#12 AND(bAHU2_Error, AHU3_DcsOccupied)
	#13 OR(#12, #15)
	#14 S bAHU1_Relay <= #16
	#15 AND(bAHU3_Error, AHU2_DcsOccupied)
	#16 AND(#13, NOT bAHU1_Relay, NOT bAHU1_Error)
	#17 R bAHU1_Relay <= #5.Q
	#18 AND(bAHU1_Trip, bAHU1_Relay)
	#19 Status_timer_1:TON(IN: #18, PT: T#2s)
	#20 AHU1_TripError <= #19.Q
	#21 AHU1_Reset:TON(IN: #9, PT: T#3s)
	#22 R bAHU1_Relay <= #21.Q
END_MACRO
#23 MACRO AHU2()
	#24 AND(bAHU2_Relay, NOT bAHU2_Error)
	#25 AHU2_DcsOccupied <= #24
	#26 OnRtrigAHU2:R_TRIG(CLK: bAHU2_On)
	#27 S bAHU2_Relay <= #26.Q
	#28 OffRtrigAHU2:R_TRIG(CLK: bAHU2_Off)
	#29 AND(NOT bAHU2_Status, bAHU2_Relay)
	#30 Status_timer_2:TON(IN: #29, PT: T#2s)
	#31 AHU2_StatusError <= #30.Q
	#32 OR(AHU2_StatusError, AHU2_TripError)
	#33 bAHU2_Error <= #34.Q
	#34 Error_timer_2:TOF(IN: #32, PT: T#5s)
	#35 AND(bAHU1_Error, AHU3_DcsOccupied)
	#36 OR(#35, #38)
	#37 S bAHU2_Relay <= #39
	#38 AND(bAHU3_Error, AHU1_DcsOccupied)
	#39 AND(#36, NOT bAHU2_Relay, NOT bAHU2_Error)
	#40 R bAHU2_Relay <= #28.Q
	#41 AND(bAHU2_Trip, bAHU2_Relay)
	#42 Status_timer_2:TON(IN: #41, PT: T#2s)
	#43 AHU2_TripError <= #42.Q
	#44 AHU2_Reset:TON(IN: #32, PT: T#3s)
	#45 R bAHU2_Relay <= #44.Q
END_MACRO
#46 MACRO AHU3()
	#47 AHU3_DcsOccupied <= #48
	#48 AND(bAHU3_Relay, NOT bAHU3_Error)
	#49 OnRtrigAHU3:R_TRIG(CLK: bAHU3_On)
	#50 S bAHU3_Relay <= #49.Q
	#51 OffRtrigAHU3:R_TRIG(CLK: bAHU3_Off)
	#52 AND(NOT bAHU3_Status, bAHU3_Relay)
	#53 Status_timer_3:TON(IN: #52, PT: T#2s)
	#54 AHU3_StatusError <= #53.Q
	#55 OR(AHU3_StatusError, AHU3_TripError)
	#56 bAHU3_Error <= #57.Q
	#57 Error_timer_3:TOF(IN: #55, PT: T#5s)
	#58 AND(bAHU1_Error, AHU2_DcsOccupied)
	#59 OR(#58, #61)
	#60 S bAHU3_Relay <= #62
	#61 AND(bAHU2_Error, AHU1_DcsOccupied)
	#62 AND(#59, NOT bAHU3_Relay, NOT bAHU3_Error)
	#63 R bAHU3_Relay <= #51.Q
	#64 AND(bAHU3_Trip, bAHU3_Relay)
	#65 Status_timer_3:TON(IN: #64, PT: T#2s)
	#66 AHU3_TripError <= #65.Q
	#67 AHU3_Reset:TON(IN: #55, PT: T#3s)
	#68 R bAHU3_Relay <= #67.Q
END_MACRO
_END_CFC_
(* the same logic as Structured Text *)
(* macro AHU1 *)
AHU1_DcsOccupied := bAHU1_Relay AND NOT bAHU1_Error;
OnRtrigAHU1(CLK := bAHU1_On);
IF OnRtrigAHU1.Q THEN bAHU1_Relay := TRUE; END_IF;
OffRtrigAHU1(CLK := bAHU1_Off);
Status_timer_1(IN := NOT bAHU1_Status AND bAHU1_Relay, PT := T#2s);
AHU1_StatusError := Status_timer_1.Q;
_t14 := AHU1_StatusError OR AHU1_TripError;
bAHU1_Error := Error_timer_1.Q;
Error_timer_1(IN := _t14, PT := T#5s);
_t34 := (bAHU2_Error AND AHU3_DcsOccupied) OR _t31;
IF _t65 THEN bAHU1_Relay := TRUE; END_IF;
_t31 := bAHU3_Error AND AHU2_DcsOccupied;
_t65 := _t34 AND NOT bAHU1_Relay AND NOT bAHU1_Error;
IF OffRtrigAHU1.Q THEN bAHU1_Relay := FALSE; END_IF;
Status_timer_1(IN := bAHU1_Trip AND bAHU1_Relay, PT := T#2s);
AHU1_TripError := Status_timer_1.Q;
AHU1_Reset(IN := _t14, PT := T#3s);
IF AHU1_Reset.Q THEN bAHU1_Relay := FALSE; END_IF;
(* macro AHU2 *)
AHU2_DcsOccupied := bAHU2_Relay AND NOT bAHU2_Error;
OnRtrigAHU2(CLK := bAHU2_On);
IF OnRtrigAHU2.Q THEN bAHU2_Relay := TRUE; END_IF;
OffRtrigAHU2(CLK := bAHU2_Off);
Status_timer_2(IN := NOT bAHU2_Status AND bAHU2_Relay, PT := T#2s);
AHU2_StatusError := Status_timer_2.Q;
_t137 := AHU2_StatusError OR AHU2_TripError;
bAHU2_Error := Error_timer_2.Q;
Error_timer_2(IN := _t137, PT := T#5s);
_t147 := (bAHU1_Error AND AHU3_DcsOccupied) OR _t150;
IF _t152 THEN bAHU2_Relay := TRUE; END_IF;
_t150 := bAHU3_Error AND AHU1_DcsOccupied;
_t152 := _t147 AND NOT bAHU2_Relay AND NOT bAHU2_Error;
IF OffRtrigAHU2.Q THEN bAHU2_Relay := FALSE; END_IF;
Status_timer_2(IN := bAHU2_Trip AND bAHU2_Relay, PT := T#2s);
AHU2_TripError := Status_timer_2.Q;
AHU2_Reset(IN := _t137, PT := T#3s);
IF AHU2_Reset.Q THEN bAHU2_Relay := FALSE; END_IF;
(* macro AHU3 *)
AHU3_DcsOccupied := _t208;
_t208 := bAHU3_Relay AND NOT bAHU3_Error;
OnRtrigAHU3(CLK := bAHU3_On);
IF OnRtrigAHU3.Q THEN bAHU3_Relay := TRUE; END_IF;
OffRtrigAHU3(CLK := bAHU3_Off);
Status_timer_3(IN := NOT bAHU3_Status AND bAHU3_Relay, PT := T#2s);
AHU3_StatusError := Status_timer_3.Q;
_t176 := AHU3_StatusError OR AHU3_TripError;
bAHU3_Error := Error_timer_3.Q;
Error_timer_3(IN := _t176, PT := T#5s);
_t186 := (bAHU1_Error AND AHU2_DcsOccupied) OR _t189;
IF _t191 THEN bAHU3_Relay := TRUE; END_IF;
_t189 := bAHU2_Error AND AHU1_DcsOccupied;
_t191 := _t186 AND NOT bAHU3_Relay AND NOT bAHU3_Error;
IF OffRtrigAHU3.Q THEN bAHU3_Relay := FALSE; END_IF;
Status_timer_3(IN := bAHU3_Trip AND bAHU3_Relay, PT := T#2s);
AHU3_TripError := Status_timer_3.Q;
AHU3_Reset(IN := _t176, PT := T#3s);
IF AHU3_Reset.Q THEN bAHU3_Relay := FALSE; END_IF;
END_FUNCTION_BLOCK

(* POU GarbageCan/Flowchart_1_2_CTRL_2, CFC *)
FUNCTION_BLOCK Flowchart_1_2_CTRL_2
VAR
	DEV_1: AHU_INTERNAL;
	DEV_2: AHU_INTERNAL;

	DEV1_ErrorInternal_1: ERROR_INTERNAL;
	DEV1_ErrorInternal_2: ERROR_INTERNAL;

	DEV2_ErrorInternal_1: ERROR_INTERNAL;
	DEV2_ErrorInternal_2: ERROR_INTERNAL;

END_VAR
VAR_INPUT
	ON1: BOOL;
	ON2: BOOL;
	ON3: BOOL;

	status_error_1 : BOOL;
	status_error_2 : BOOL;
	status_error_3 : BOOL;

	trip_error_1 : BOOL;
	trip_error_2 : BOOL;
	trip_error_3 : BOOL;


END_VAR
VAR_IN_OUT
	Latch1:BOOL;
	Latch2:BOOL;
	Latch3:BOOL;
END_VAR
VAR_OUTPUT
	DcsOccupied_1: BOOL;
	DcsOccupied_2: BOOL;
	DcsOccupied_3: BOOL;
END_VAR
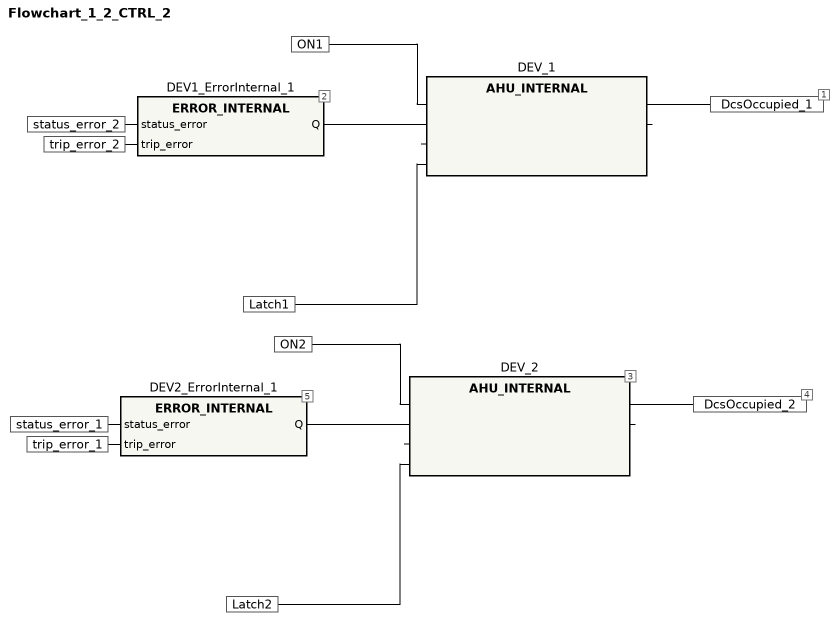
_CFC_ (* Continuous Function Chart, elements in execution order *)
#0 DEV_1:AHU_INTERNAL(ON1, #2.Q, -, Latch1)
#1 DcsOccupied_1 <= #0.out 1
#2 DEV1_ErrorInternal_1:ERROR_INTERNAL(status_error: status_error_2, trip_error: trip_error_2)
#3 DEV_2:AHU_INTERNAL(ON2, #5.Q, -, Latch2)
#4 DcsOccupied_2 <= #3.out 1
#5 DEV2_ErrorInternal_1:ERROR_INTERNAL(status_error: status_error_1, trip_error: trip_error_1)
_END_CFC_
END_FUNCTION_BLOCK

(* POU GarbageCan/Flowchart_3_4, CFC *)
FUNCTION_BLOCK Flowchart_3_4
VAR_INPUT
	bAHU1_On: BOOL;
	bAHU1_Off: BOOL;


	bAHU2_On: BOOL;
	bAHU2_Off: BOOL;

END_VAR
VAR_OUTPUT
	AHU1_DcsOccupied AT%Q*: BOOL;
	AHU1_StatusError  AT%Q*: BOOL;
	AHU1_TripError AT%Q*: BOOL;

	AHU2_DcsOccupied AT%Q*: BOOL;
	AHU2_StatusError  AT%Q*: BOOL;
	AHU2_TripError AT%Q*: BOOL;

END_VAR
VAR

	bAHU1_Error: BOOL;
	bAHU2_Error: BOOL;

	bAHU1_Status AT %I*: BOOL;
	bAHU1_Trip AT %I*: BOOL;
	bAHU1_Relay AT %Q*: BOOL;
	Status_timer_1: TON;
	Error_timer_1: TOF;
	OnRtrigAHU1: R_TRIG;
	OffRtrigAHU1: R_TRIG;


	bAHU2_Status AT %I*: BOOL;
	bAHU2_Trip AT %I*: BOOL;
	bAHU2_Relay AT %Q*: BOOL;
	Status_timer_2: TON;
	Error_timer_2: TOF;
	OnRtrigAHU2: R_TRIG;
	OffRtrigAHU2: R_TRIG;


	AHU1_Reset: TON;
	AHU2_Reset: TON;
END_VAR
VAR (* helpers for the ST form of the networks *)
	_t14 : BOOL;
	_t65 : BOOL;
	_t137 : BOOL;
	_t152 : BOOL;
END_VAR
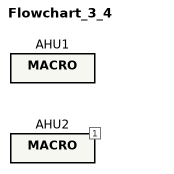
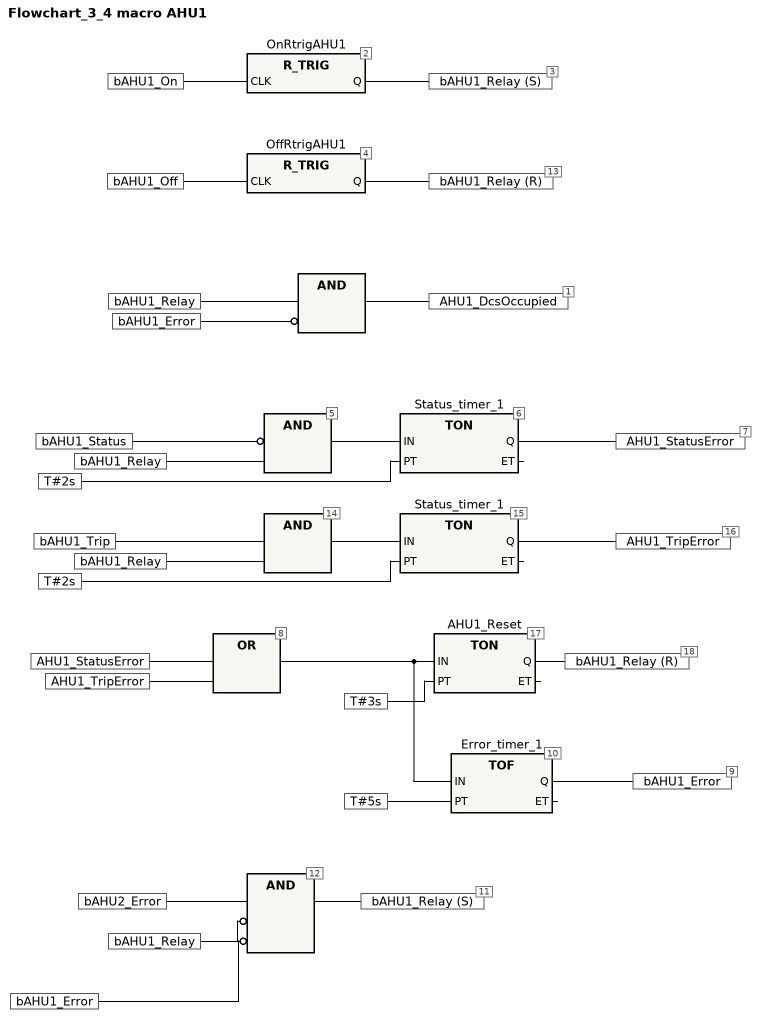
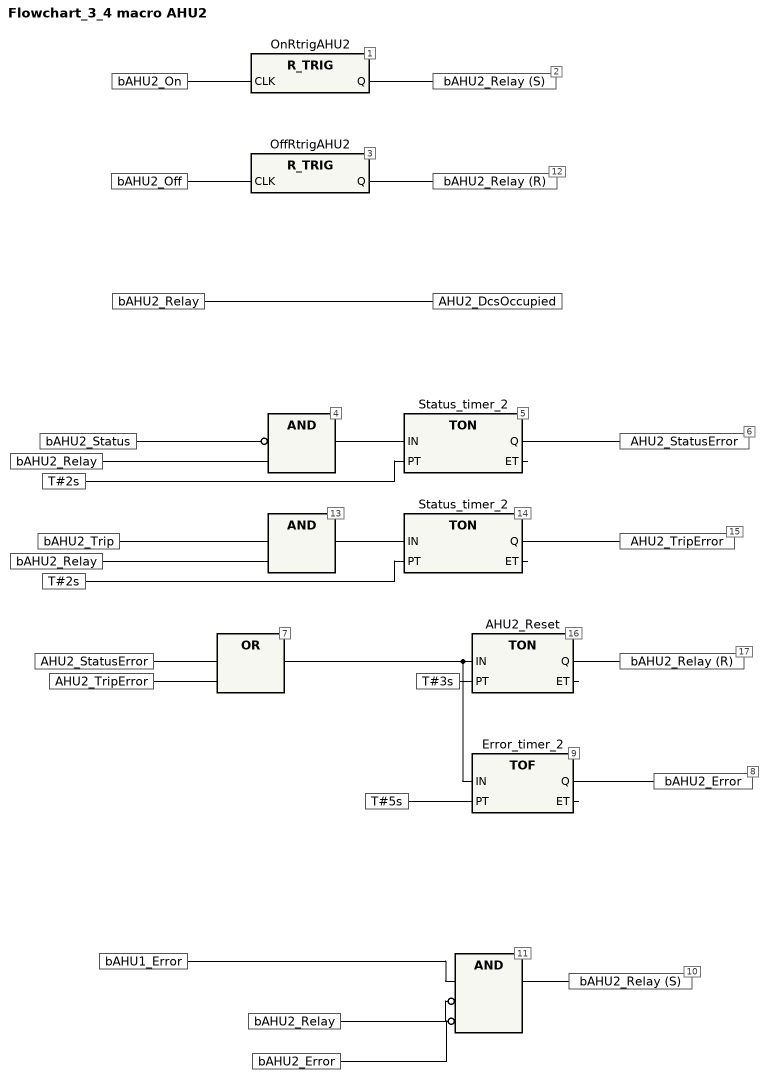
_CFC_ (* Continuous Function Chart, elements in execution order *)
#0 MACRO AHU1()
	#1 AND(bAHU1_Relay, NOT bAHU1_Error)
	#2 AHU1_DcsOccupied <= #1
	#3 OnRtrigAHU1:R_TRIG(CLK: bAHU1_On)
	#4 S bAHU1_Relay <= #3.Q
	#5 OffRtrigAHU1:R_TRIG(CLK: bAHU1_Off)
	#6 AND(NOT bAHU1_Status, bAHU1_Relay)
	#7 Status_timer_1:TON(IN: #6, PT: T#2s)
	#8 AHU1_StatusError <= #7.Q
	#9 OR(AHU1_StatusError, AHU1_TripError)
	#10 bAHU1_Error <= #11.Q
	#11 Error_timer_1:TOF(IN: #9, PT: T#5s)
	#12 S bAHU1_Relay <= #13
	#13 AND(bAHU2_Error, NOT bAHU1_Relay, NOT bAHU1_Error)
	#14 R bAHU1_Relay <= #5.Q
	#15 AND(bAHU1_Trip, bAHU1_Relay)
	#16 Status_timer_1:TON(IN: #15, PT: T#2s)
	#17 AHU1_TripError <= #16.Q
	#18 AHU1_Reset:TON(IN: #9, PT: T#3s)
	#19 R bAHU1_Relay <= #18.Q
END_MACRO
#20 MACRO AHU2()
	#21 AHU2_DcsOccupied <= bAHU2_Relay
	#22 OnRtrigAHU2:R_TRIG(CLK: bAHU2_On)
	#23 S bAHU2_Relay <= #22.Q
	#24 OffRtrigAHU2:R_TRIG(CLK: bAHU2_Off)
	#25 AND(NOT bAHU2_Status, bAHU2_Relay)
	#26 Status_timer_2:TON(IN: #25, PT: T#2s)
	#27 AHU2_StatusError <= #26.Q
	#28 OR(AHU2_StatusError, AHU2_TripError)
	#29 bAHU2_Error <= #30.Q
	#30 Error_timer_2:TOF(IN: #28, PT: T#5s)
	#31 S bAHU2_Relay <= #32
	#32 AND(bAHU1_Error, NOT bAHU2_Relay, NOT bAHU2_Error)
	#33 R bAHU2_Relay <= #24.Q
	#34 AND(bAHU2_Trip, bAHU2_Relay)
	#35 Status_timer_2:TON(IN: #34, PT: T#2s)
	#36 AHU2_TripError <= #35.Q
	#37 AHU2_Reset:TON(IN: #28, PT: T#3s)
	#38 R bAHU2_Relay <= #37.Q
END_MACRO
_END_CFC_
(* the same logic as Structured Text *)
(* macro AHU1 *)
AHU1_DcsOccupied := bAHU1_Relay AND NOT bAHU1_Error;
OnRtrigAHU1(CLK := bAHU1_On);
IF OnRtrigAHU1.Q THEN bAHU1_Relay := TRUE; END_IF;
OffRtrigAHU1(CLK := bAHU1_Off);
Status_timer_1(IN := NOT bAHU1_Status AND bAHU1_Relay, PT := T#2s);
AHU1_StatusError := Status_timer_1.Q;
_t14 := AHU1_StatusError OR AHU1_TripError;
bAHU1_Error := Error_timer_1.Q;
Error_timer_1(IN := _t14, PT := T#5s);
IF _t65 THEN bAHU1_Relay := TRUE; END_IF;
_t65 := bAHU2_Error AND NOT bAHU1_Relay AND NOT bAHU1_Error;
IF OffRtrigAHU1.Q THEN bAHU1_Relay := FALSE; END_IF;
Status_timer_1(IN := bAHU1_Trip AND bAHU1_Relay, PT := T#2s);
AHU1_TripError := Status_timer_1.Q;
AHU1_Reset(IN := _t14, PT := T#3s);
IF AHU1_Reset.Q THEN bAHU1_Relay := FALSE; END_IF;
(* macro AHU2 *)
AHU2_DcsOccupied := bAHU2_Relay;
OnRtrigAHU2(CLK := bAHU2_On);
IF OnRtrigAHU2.Q THEN bAHU2_Relay := TRUE; END_IF;
OffRtrigAHU2(CLK := bAHU2_Off);
Status_timer_2(IN := NOT bAHU2_Status AND bAHU2_Relay, PT := T#2s);
AHU2_StatusError := Status_timer_2.Q;
_t137 := AHU2_StatusError OR AHU2_TripError;
bAHU2_Error := Error_timer_2.Q;
Error_timer_2(IN := _t137, PT := T#5s);
IF _t152 THEN bAHU2_Relay := TRUE; END_IF;
_t152 := bAHU1_Error AND NOT bAHU2_Relay AND NOT bAHU2_Error;
IF OffRtrigAHU2.Q THEN bAHU2_Relay := FALSE; END_IF;
Status_timer_2(IN := bAHU2_Trip AND bAHU2_Relay, PT := T#2s);
AHU2_TripError := Status_timer_2.Q;
AHU2_Reset(IN := _t137, PT := T#3s);
IF AHU2_Reset.Q THEN bAHU2_Relay := FALSE; END_IF;
END_FUNCTION_BLOCK
